(* Logix 5000 project; controller reports 1756-L63 rev 20.15; software revision 20.04; part 29 of 52 *)

        [2115].log_data[19].valid := 1, [2115].time.Year := 2023, [2115].time.Month := 1, [2115].time.Day := 17, [2115].time.Minute := 39, [2115].time.Second := 59, [2116].log_data[0].min := 1.0, [2116].log_data[0].max := 1.0, [2116].log_data[0].total := 300.0, [2116].log_data[0].time := 300.0, [2116].log_data[0].minminute := 40, [2116].log_data[0].maxminute := 40, [2116].log_data[0].valid := 1, [2116].log_data[1].valid := 1, [2116].log_data[2].valid := 1, [2116].log_data[3].valid := 1, [2116].log_data[4].valid := 1, [2116].log_data[5].valid := 1, [2116].log_data[6].valid := 1, [2116].log_data[7].valid := 1, [2116].log_data[8].valid := 1, [2116].log_data[9].valid := 1, [2116].log_data[10].valid := 1, [2116].log_data[11].valid := 1, [2116].log_data[12].valid := 1, [2116].log_data[13].valid := 1, [2116].log_data[14].valid := 1, [2116].log_data[15].valid := 1, [2116].log_data[16].valid := 1, [2116].log_data[17].valid := 1, [2116].log_data[18].valid := 1, [2116].log_data[19].valid := 1, [2116].time.Year := 2023, [2116].time.Month := 1, [2116].time.Day := 17, [2116].time.Minute := 44, [2116].time.Second := 59, [2117].log_data[0].min := 1.0, [2117].log_data[0].max := 1.0, [2117].log_data[0].total := 300.0, [2117].log_data[0].time := 300.0, [2117].log_data[0].minminute := 45, [2117].log_data[0].maxminute := 45, [2117].log_data[0].valid := 1, [2117].log_data[1].valid := 1, [2117].log_data[2].valid := 1, [2117].log_data[3].valid := 1, [2117].log_data[4].valid := 1, [2117].log_data[5].valid := 1, [2117].log_data[6].valid := 1, [2117].log_data[7].valid := 1, [2117].log_data[8].valid := 1, [2117].log_data[9].valid := 1, [2117].log_data[10].valid := 1, [2117].log_data[11].valid := 1, [2117].log_data[12].valid := 1, [2117].log_data[13].valid := 1, [2117].log_data[14].valid := 1, [2117].log_data[15].valid := 1, [2117].log_data[16].valid := 1,
        [2117].log_data[17].valid := 1, [2117].log_data[18].valid := 1, [2117].log_data[19].valid := 1, [2117].time.Year := 2023, [2117].time.Month := 1, [2117].time.Day := 17, [2117].time.Minute := 49, [2117].time.Second := 59, [2118].log_data[0].min := 1.0, [2118].log_data[0].max := 1.0, [2118].log_data[0].total := 300.0, [2118].log_data[0].time := 300.0, [2118].log_data[0].minminute := 50, [2118].log_data[0].maxminute := 50, [2118].log_data[0].valid := 1, [2118].log_data[1].valid := 1, [2118].log_data[2].valid := 1, [2118].log_data[3].valid := 1, [2118].log_data[4].valid := 1, [2118].log_data[5].valid := 1, [2118].log_data[6].valid := 1, [2118].log_data[7].valid := 1, [2118].log_data[8].valid := 1, [2118].log_data[9].valid := 1, [2118].log_data[10].valid := 1, [2118].log_data[11].valid := 1, [2118].log_data[12].valid := 1, [2118].log_data[13].valid := 1, [2118].log_data[14].valid := 1, [2118].log_data[15].valid := 1, [2118].log_data[16].valid := 1, [2118].log_data[17].valid := 1, [2118].log_data[18].valid := 1, [2118].log_data[19].valid := 1, [2118].time.Year := 2023, [2118].time.Month := 1, [2118].time.Day := 17, [2118].time.Minute := 54, [2118].time.Second := 59, [2119].log_data[0].min := 1.0, [2119].log_data[0].max := 1.0, [2119].log_data[0].total := 300.0, [2119].log_data[0].time := 300.0, [2119].log_data[0].minminute := 55, [2119].log_data[0].maxminute := 55, [2119].log_data[0].valid := 1, [2119].log_data[1].valid := 1, [2119].log_data[2].valid := 1, [2119].log_data[3].valid := 1, [2119].log_data[4].valid := 1, [2119].log_data[5].valid := 1, [2119].log_data[6].valid := 1, [2119].log_data[7].valid := 1, [2119].log_data[8].valid := 1, [2119].log_data[9].valid := 1, [2119].log_data[10].valid := 1, [2119].log_data[11].valid := 1, [2119].log_data[12].valid := 1, [2119].log_data[13].valid := 1, [2119].log_data[14].valid := 1,
        [2119].log_data[15].valid := 1, [2119].log_data[16].valid := 1, [2119].log_data[17].valid := 1, [2119].log_data[18].valid := 1, [2119].log_data[19].valid := 1, [2119].time.Year := 2023, [2119].time.Month := 1, [2119].time.Day := 17, [2119].time.Minute := 59, [2119].time.Second := 59, [2120].log_data[0].min := 1.0, [2120].log_data[0].max := 1.0, [2120].log_data[0].total := 300.0, [2120].log_data[0].time := 300.0, [2120].log_data[0].valid := 1, [2120].log_data[1].valid := 1, [2120].log_data[2].valid := 1, [2120].log_data[3].valid := 1, [2120].log_data[4].valid := 1, [2120].log_data[5].valid := 1, [2120].log_data[6].valid := 1, [2120].log_data[7].valid := 1, [2120].log_data[8].valid := 1, [2120].log_data[9].valid := 1, [2120].log_data[10].valid := 1, [2120].log_data[11].valid := 1, [2120].log_data[12].valid := 1, [2120].log_data[13].valid := 1, [2120].log_data[14].valid := 1, [2120].log_data[15].valid := 1, [2120].log_data[16].valid := 1, [2120].log_data[17].valid := 1, [2120].log_data[18].valid := 1, [2120].log_data[19].valid := 1, [2120].time.Year := 2023, [2120].time.Month := 1, [2120].time.Day := 17, [2120].time.Hour := 1, [2120].time.Minute := 4, [2120].time.Second := 59, [2121].log_data[0].min := 1.0, [2121].log_data[0].max := 1.0, [2121].log_data[0].total := 300.0, [2121].log_data[0].time := 300.0, [2121].log_data[0].minminute := 5, [2121].log_data[0].maxminute := 5, [2121].log_data[0].valid := 1, [2121].log_data[1].valid := 1, [2121].log_data[2].valid := 1, [2121].log_data[3].valid := 1, [2121].log_data[4].valid := 1, [2121].log_data[5].valid := 1, [2121].log_data[6].valid := 1, [2121].log_data[7].valid := 1, [2121].log_data[8].valid := 1, [2121].log_data[9].valid := 1, [2121].log_data[10].valid := 1, [2121].log_data[11].valid := 1, [2121].log_data[12].valid := 1, [2121].log_data[13].valid := 1,
        [2121].log_data[14].valid := 1, [2121].log_data[15].valid := 1, [2121].log_data[16].valid := 1, [2121].log_data[17].valid := 1, [2121].log_data[18].valid := 1, [2121].log_data[19].valid := 1, [2121].time.Year := 2023, [2121].time.Month := 1, [2121].time.Day := 17, [2121].time.Hour := 1, [2121].time.Minute := 9, [2121].time.Second := 59, [2122].log_data[0].min := 1.0, [2122].log_data[0].max := 1.0, [2122].log_data[0].total := 300.0, [2122].log_data[0].time := 300.0, [2122].log_data[0].minminute := 10, [2122].log_data[0].maxminute := 10, [2122].log_data[0].valid := 1, [2122].log_data[1].valid := 1, [2122].log_data[2].valid := 1, [2122].log_data[3].valid := 1, [2122].log_data[4].valid := 1, [2122].log_data[5].valid := 1, [2122].log_data[6].valid := 1, [2122].log_data[7].valid := 1, [2122].log_data[8].valid := 1, [2122].log_data[9].valid := 1, [2122].log_data[10].valid := 1, [2122].log_data[11].valid := 1, [2122].log_data[12].valid := 1, [2122].log_data[13].valid := 1, [2122].log_data[14].valid := 1, [2122].log_data[15].valid := 1, [2122].log_data[16].valid := 1, [2122].log_data[17].valid := 1, [2122].log_data[18].valid := 1, [2122].log_data[19].valid := 1, [2122].time.Year := 2023, [2122].time.Month := 1, [2122].time.Day := 17, [2122].time.Hour := 1, [2122].time.Minute := 14, [2122].time.Second := 59, [2123].log_data[0].min := 1.0, [2123].log_data[0].max := 1.0, [2123].log_data[0].total := 300.0, [2123].log_data[0].time := 300.0, [2123].log_data[0].minminute := 15, [2123].log_data[0].maxminute := 15, [2123].log_data[0].valid := 1, [2123].log_data[1].valid := 1, [2123].log_data[2].valid := 1, [2123].log_data[3].valid := 1, [2123].log_data[4].valid := 1, [2123].log_data[5].valid := 1, [2123].log_data[6].valid := 1, [2123].log_data[7].valid := 1, [2123].log_data[8].valid := 1, [2123].log_data[9].valid := 1,
        [2123].log_data[10].valid := 1, [2123].log_data[11].valid := 1, [2123].log_data[12].valid := 1, [2123].log_data[13].valid := 1, [2123].log_data[14].valid := 1, [2123].log_data[15].valid := 1, [2123].log_data[16].valid := 1, [2123].log_data[17].valid := 1, [2123].log_data[18].valid := 1, [2123].log_data[19].valid := 1, [2123].time.Year := 2023, [2123].time.Month := 1, [2123].time.Day := 17, [2123].time.Hour := 1, [2123].time.Minute := 19, [2123].time.Second := 59, [2124].log_data[0].min := 1.0, [2124].log_data[0].max := 1.0, [2124].log_data[0].total := 300.0, [2124].log_data[0].time := 300.0, [2124].log_data[0].minminute := 20, [2124].log_data[0].maxminute := 20, [2124].log_data[0].valid := 1, [2124].log_data[1].valid := 1, [2124].log_data[2].valid := 1, [2124].log_data[3].valid := 1, [2124].log_data[4].valid := 1, [2124].log_data[5].valid := 1, [2124].log_data[6].valid := 1, [2124].log_data[7].valid := 1, [2124].log_data[8].valid := 1, [2124].log_data[9].valid := 1, [2124].log_data[10].valid := 1, [2124].log_data[11].valid := 1, [2124].log_data[12].valid := 1, [2124].log_data[13].valid := 1, [2124].log_data[14].valid := 1, [2124].log_data[15].valid := 1, [2124].log_data[16].valid := 1, [2124].log_data[17].valid := 1, [2124].log_data[18].valid := 1, [2124].log_data[19].valid := 1, [2124].time.Year := 2023, [2124].time.Month := 1, [2124].time.Day := 17, [2124].time.Hour := 1, [2124].time.Minute := 24, [2124].time.Second := 59, [2125].log_data[0].min := 1.0, [2125].log_data[0].max := 1.0, [2125].log_data[0].total := 300.0, [2125].log_data[0].time := 300.0, [2125].log_data[0].minminute := 25, [2125].log_data[0].maxminute := 25, [2125].log_data[0].valid := 1, [2125].log_data[1].valid := 1, [2125].log_data[2].valid := 1, [2125].log_data[3].valid := 1, [2125].log_data[4].valid := 1, [2125].log_data[5].valid := 1,
        [2125].log_data[6].valid := 1, [2125].log_data[7].valid := 1, [2125].log_data[8].valid := 1, [2125].log_data[9].valid := 1, [2125].log_data[10].valid := 1, [2125].log_data[11].valid := 1, [2125].log_data[12].valid := 1, [2125].log_data[13].valid := 1, [2125].log_data[14].valid := 1, [2125].log_data[15].valid := 1, [2125].log_data[16].valid := 1, [2125].log_data[17].valid := 1, [2125].log_data[18].valid := 1, [2125].log_data[19].valid := 1, [2125].time.Year := 2023, [2125].time.Month := 1, [2125].time.Day := 17, [2125].time.Hour := 1, [2125].time.Minute := 29, [2125].time.Second := 59, [2126].log_data[0].min := 1.0, [2126].log_data[0].max := 1.0, [2126].log_data[0].total := 300.0, [2126].log_data[0].time := 300.0, [2126].log_data[0].minminute := 30, [2126].log_data[0].maxminute := 30, [2126].log_data[0].valid := 1, [2126].log_data[1].valid := 1, [2126].log_data[2].valid := 1, [2126].log_data[3].valid := 1, [2126].log_data[4].valid := 1, [2126].log_data[5].valid := 1, [2126].log_data[6].valid := 1, [2126].log_data[7].valid := 1, [2126].log_data[8].valid := 1, [2126].log_data[9].valid := 1, [2126].log_data[10].valid := 1, [2126].log_data[11].valid := 1, [2126].log_data[12].valid := 1, [2126].log_data[13].valid := 1, [2126].log_data[14].valid := 1, [2126].log_data[15].valid := 1, [2126].log_data[16].valid := 1, [2126].log_data[17].valid := 1, [2126].log_data[18].valid := 1, [2126].log_data[19].valid := 1, [2126].time.Year := 2023, [2126].time.Month := 1, [2126].time.Day := 17, [2126].time.Hour := 1, [2126].time.Minute := 34, [2126].time.Second := 59, [2127].log_data[0].min := 1.0, [2127].log_data[0].max := 1.0, [2127].log_data[0].total := 300.0, [2127].log_data[0].time := 300.0, [2127].log_data[0].minminute := 35, [2127].log_data[0].maxminute := 35, [2127].log_data[0].valid := 1, [2127].log_data[1].valid := 1,
        [2127].log_data[2].valid := 1, [2127].log_data[3].valid := 1, [2127].log_data[4].valid := 1, [2127].log_data[5].valid := 1, [2127].log_data[6].valid := 1, [2127].log_data[7].valid := 1, [2127].log_data[8].valid := 1, [2127].log_data[9].valid := 1, [2127].log_data[10].valid := 1, [2127].log_data[11].valid := 1, [2127].log_data[12].valid := 1, [2127].log_data[13].valid := 1, [2127].log_data[14].valid := 1, [2127].log_data[15].valid := 1, [2127].log_data[16].valid := 1, [2127].log_data[17].valid := 1, [2127].log_data[18].valid := 1, [2127].log_data[19].valid := 1, [2127].time.Year := 2023, [2127].time.Month := 1, [2127].time.Day := 17, [2127].time.Hour := 1, [2127].time.Minute := 39, [2127].time.Second := 59, [2128].log_data[0].min := 1.0, [2128].log_data[0].max := 1.0, [2128].log_data[0].total := 300.0, [2128].log_data[0].time := 300.0, [2128].log_data[0].minminute := 40, [2128].log_data[0].maxminute := 40, [2128].log_data[0].valid := 1, [2128].log_data[1].valid := 1, [2128].log_data[2].valid := 1, [2128].log_data[3].valid := 1, [2128].log_data[4].valid := 1, [2128].log_data[5].valid := 1, [2128].log_data[6].valid := 1, [2128].log_data[7].valid := 1, [2128].log_data[8].valid := 1, [2128].log_data[9].valid := 1, [2128].log_data[10].valid := 1, [2128].log_data[11].valid := 1, [2128].log_data[12].valid := 1, [2128].log_data[13].valid := 1, [2128].log_data[14].valid := 1, [2128].log_data[15].valid := 1, [2128].log_data[16].valid := 1, [2128].log_data[17].valid := 1, [2128].log_data[18].valid := 1, [2128].log_data[19].valid := 1, [2128].time.Year := 2023, [2128].time.Month := 1, [2128].time.Day := 17, [2128].time.Hour := 1, [2128].time.Minute := 44, [2128].time.Second := 59, [2129].log_data[0].min := 1.0, [2129].log_data[0].max := 1.0, [2129].log_data[0].total := 300.0, [2129].log_data[0].time := 300.0,
        [2129].log_data[0].minminute := 45, [2129].log_data[0].maxminute := 45, [2129].log_data[0].valid := 1, [2129].log_data[1].valid := 1, [2129].log_data[2].valid := 1, [2129].log_data[3].valid := 1, [2129].log_data[4].valid := 1, [2129].log_data[5].valid := 1, [2129].log_data[6].valid := 1, [2129].log_data[7].valid := 1, [2129].log_data[8].valid := 1, [2129].log_data[9].valid := 1, [2129].log_data[10].valid := 1, [2129].log_data[11].valid := 1, [2129].log_data[12].valid := 1, [2129].log_data[13].valid := 1, [2129].log_data[14].valid := 1, [2129].log_data[15].valid := 1, [2129].log_data[16].valid := 1, [2129].log_data[17].valid := 1, [2129].log_data[18].valid := 1, [2129].log_data[19].valid := 1, [2129].time.Year := 2023, [2129].time.Month := 1, [2129].time.Day := 17, [2129].time.Hour := 1, [2129].time.Minute := 49, [2129].time.Second := 59, [2130].log_data[0].min := 1.0, [2130].log_data[0].max := 1.0, [2130].log_data[0].total := 300.0, [2130].log_data[0].time := 300.0, [2130].log_data[0].minminute := 50, [2130].log_data[0].maxminute := 50, [2130].log_data[0].valid := 1, [2130].log_data[1].valid := 1, [2130].log_data[2].valid := 1, [2130].log_data[3].valid := 1, [2130].log_data[4].valid := 1, [2130].log_data[5].valid := 1, [2130].log_data[6].valid := 1, [2130].log_data[7].valid := 1, [2130].log_data[8].valid := 1, [2130].log_data[9].valid := 1, [2130].log_data[10].valid := 1, [2130].log_data[11].valid := 1, [2130].log_data[12].valid := 1, [2130].log_data[13].valid := 1, [2130].log_data[14].valid := 1, [2130].log_data[15].valid := 1, [2130].log_data[16].valid := 1, [2130].log_data[17].valid := 1, [2130].log_data[18].valid := 1, [2130].log_data[19].valid := 1, [2130].time.Year := 2023, [2130].time.Month := 1, [2130].time.Day := 17, [2130].time.Hour := 1, [2130].time.Minute := 54, [2130].time.Second := 59,
        [2131].log_data[0].min := 1.0, [2131].log_data[0].max := 1.0, [2131].log_data[0].total := 300.0, [2131].log_data[0].time := 300.0, [2131].log_data[0].minminute := 55, [2131].log_data[0].maxminute := 55, [2131].log_data[0].valid := 1, [2131].log_data[1].valid := 1, [2131].log_data[2].valid := 1, [2131].log_data[3].valid := 1, [2131].log_data[4].valid := 1, [2131].log_data[5].valid := 1, [2131].log_data[6].valid := 1, [2131].log_data[7].valid := 1, [2131].log_data[8].valid := 1, [2131].log_data[9].valid := 1, [2131].log_data[10].valid := 1, [2131].log_data[11].valid := 1, [2131].log_data[12].valid := 1, [2131].log_data[13].valid := 1, [2131].log_data[14].valid := 1, [2131].log_data[15].valid := 1, [2131].log_data[16].valid := 1, [2131].log_data[17].valid := 1, [2131].log_data[18].valid := 1, [2131].log_data[19].valid := 1, [2131].time.Year := 2023, [2131].time.Month := 1, [2131].time.Day := 17, [2131].time.Hour := 1, [2131].time.Minute := 59, [2131].time.Second := 59, [2132].log_data[0].min := 1.0, [2132].log_data[0].max := 1.0, [2132].log_data[0].total := 300.0, [2132].log_data[0].time := 300.0, [2132].log_data[0].valid := 1, [2132].log_data[1].valid := 1, [2132].log_data[2].valid := 1, [2132].log_data[3].valid := 1, [2132].log_data[4].valid := 1, [2132].log_data[5].valid := 1, [2132].log_data[6].valid := 1, [2132].log_data[7].valid := 1, [2132].log_data[8].valid := 1, [2132].log_data[9].valid := 1, [2132].log_data[10].valid := 1, [2132].log_data[11].valid := 1, [2132].log_data[12].valid := 1, [2132].log_data[13].valid := 1, [2132].log_data[14].valid := 1, [2132].log_data[15].valid := 1, [2132].log_data[16].valid := 1, [2132].log_data[17].valid := 1, [2132].log_data[18].valid := 1, [2132].log_data[19].valid := 1, [2132].time.Year := 2023, [2132].time.Month := 1, [2132].time.Day := 17, [2132].time.Hour := 2,
        [2132].time.Minute := 4, [2132].time.Second := 59, [2133].log_data[0].min := 1.0, [2133].log_data[0].max := 1.0, [2133].log_data[0].total := 300.0, [2133].log_data[0].time := 300.0, [2133].log_data[0].minminute := 5, [2133].log_data[0].maxminute := 5, [2133].log_data[0].valid := 1, [2133].log_data[1].valid := 1, [2133].log_data[2].valid := 1, [2133].log_data[3].valid := 1, [2133].log_data[4].valid := 1, [2133].log_data[5].valid := 1, [2133].log_data[6].valid := 1, [2133].log_data[7].valid := 1, [2133].log_data[8].valid := 1, [2133].log_data[9].valid := 1, [2133].log_data[10].valid := 1, [2133].log_data[11].valid := 1, [2133].log_data[12].valid := 1, [2133].log_data[13].valid := 1, [2133].log_data[14].valid := 1, [2133].log_data[15].valid := 1, [2133].log_data[16].valid := 1, [2133].log_data[17].valid := 1, [2133].log_data[18].valid := 1, [2133].log_data[19].valid := 1, [2133].time.Year := 2023, [2133].time.Month := 1, [2133].time.Day := 17, [2133].time.Hour := 2, [2133].time.Minute := 9, [2133].time.Second := 59, [2134].log_data[0].min := 1.0, [2134].log_data[0].max := 1.0, [2134].log_data[0].total := 300.0, [2134].log_data[0].time := 300.0, [2134].log_data[0].minminute := 10, [2134].log_data[0].maxminute := 10, [2134].log_data[0].valid := 1, [2134].log_data[1].valid := 1, [2134].log_data[2].valid := 1, [2134].log_data[3].valid := 1, [2134].log_data[4].valid := 1, [2134].log_data[5].valid := 1, [2134].log_data[6].valid := 1, [2134].log_data[7].valid := 1, [2134].log_data[8].valid := 1, [2134].log_data[9].valid := 1, [2134].log_data[10].valid := 1, [2134].log_data[11].valid := 1, [2134].log_data[12].valid := 1, [2134].log_data[13].valid := 1, [2134].log_data[14].valid := 1, [2134].log_data[15].valid := 1, [2134].log_data[16].valid := 1, [2134].log_data[17].valid := 1, [2134].log_data[18].valid := 1, [2134].log_data[19].valid := 1,
        [2134].time.Year := 2023, [2134].time.Month := 1, [2134].time.Day := 17, [2134].time.Hour := 2, [2134].time.Minute := 14, [2134].time.Second := 59, [2135].log_data[0].min := 1.0, [2135].log_data[0].max := 1.0, [2135].log_data[0].total := 300.0, [2135].log_data[0].time := 300.0, [2135].log_data[0].minminute := 15, [2135].log_data[0].maxminute := 15, [2135].log_data[0].valid := 1, [2135].log_data[1].valid := 1, [2135].log_data[2].valid := 1, [2135].log_data[3].valid := 1, [2135].log_data[4].valid := 1, [2135].log_data[5].valid := 1, [2135].log_data[6].valid := 1, [2135].log_data[7].valid := 1, [2135].log_data[8].valid := 1, [2135].log_data[9].valid := 1, [2135].log_data[10].valid := 1, [2135].log_data[11].valid := 1, [2135].log_data[12].valid := 1, [2135].log_data[13].valid := 1, [2135].log_data[14].valid := 1, [2135].log_data[15].valid := 1, [2135].log_data[16].valid := 1, [2135].log_data[17].valid := 1, [2135].log_data[18].valid := 1, [2135].log_data[19].valid := 1, [2135].time.Year := 2023, [2135].time.Month := 1, [2135].time.Day := 17, [2135].time.Hour := 2, [2135].time.Minute := 19, [2135].time.Second := 59, [2136].log_data[0].min := 1.0, [2136].log_data[0].max := 1.0, [2136].log_data[0].total := 300.0, [2136].log_data[0].time := 300.0, [2136].log_data[0].minminute := 20, [2136].log_data[0].maxminute := 20, [2136].log_data[0].valid := 1, [2136].log_data[1].valid := 1, [2136].log_data[2].valid := 1, [2136].log_data[3].valid := 1, [2136].log_data[4].valid := 1, [2136].log_data[5].valid := 1, [2136].log_data[6].valid := 1, [2136].log_data[7].valid := 1, [2136].log_data[8].valid := 1, [2136].log_data[9].valid := 1, [2136].log_data[10].valid := 1, [2136].log_data[11].valid := 1, [2136].log_data[12].valid := 1, [2136].log_data[13].valid := 1, [2136].log_data[14].valid := 1, [2136].log_data[15].valid := 1,
        [2136].log_data[16].valid := 1, [2136].log_data[17].valid := 1, [2136].log_data[18].valid := 1, [2136].log_data[19].valid := 1, [2136].time.Year := 2023, [2136].time.Month := 1, [2136].time.Day := 17, [2136].time.Hour := 2, [2136].time.Minute := 24, [2136].time.Second := 59, [2137].log_data[0].min := 1.0, [2137].log_data[0].max := 1.0, [2137].log_data[0].total := 300.0, [2137].log_data[0].time := 300.0, [2137].log_data[0].minminute := 25, [2137].log_data[0].maxminute := 25, [2137].log_data[0].valid := 1, [2137].log_data[1].valid := 1, [2137].log_data[2].valid := 1, [2137].log_data[3].valid := 1, [2137].log_data[4].valid := 1, [2137].log_data[5].valid := 1, [2137].log_data[6].valid := 1, [2137].log_data[7].valid := 1, [2137].log_data[8].valid := 1, [2137].log_data[9].valid := 1, [2137].log_data[10].valid := 1, [2137].log_data[11].valid := 1, [2137].log_data[12].valid := 1, [2137].log_data[13].valid := 1, [2137].log_data[14].valid := 1, [2137].log_data[15].valid := 1, [2137].log_data[16].valid := 1, [2137].log_data[17].valid := 1, [2137].log_data[18].valid := 1, [2137].log_data[19].valid := 1, [2137].time.Year := 2023, [2137].time.Month := 1, [2137].time.Day := 17, [2137].time.Hour := 2, [2137].time.Minute := 29, [2137].time.Second := 59, [2138].log_data[0].min := 1.0, [2138].log_data[0].max := 1.0, [2138].log_data[0].total := 300.0, [2138].log_data[0].time := 300.0, [2138].log_data[0].minminute := 30, [2138].log_data[0].maxminute := 30, [2138].log_data[0].valid := 1, [2138].log_data[1].valid := 1, [2138].log_data[2].valid := 1, [2138].log_data[3].valid := 1, [2138].log_data[4].valid := 1, [2138].log_data[5].valid := 1, [2138].log_data[6].valid := 1, [2138].log_data[7].valid := 1, [2138].log_data[8].valid := 1, [2138].log_data[9].valid := 1, [2138].log_data[10].valid := 1, [2138].log_data[11].valid := 1,
        [2138].log_data[12].valid := 1, [2138].log_data[13].valid := 1, [2138].log_data[14].valid := 1, [2138].log_data[15].valid := 1, [2138].log_data[16].valid := 1, [2138].log_data[17].valid := 1, [2138].log_data[18].valid := 1, [2138].log_data[19].valid := 1, [2138].time.Year := 2023, [2138].time.Month := 1, [2138].time.Day := 17, [2138].time.Hour := 2, [2138].time.Minute := 34, [2138].time.Second := 59, [2139].log_data[0].min := 1.0, [2139].log_data[0].max := 1.0, [2139].log_data[0].total := 300.0, [2139].log_data[0].time := 300.0, [2139].log_data[0].minminute := 35, [2139].log_data[0].maxminute := 35, [2139].log_data[0].valid := 1, [2139].log_data[1].valid := 1, [2139].log_data[2].valid := 1, [2139].log_data[3].valid := 1, [2139].log_data[4].valid := 1, [2139].log_data[5].valid := 1, [2139].log_data[6].valid := 1, [2139].log_data[7].valid := 1, [2139].log_data[8].valid := 1, [2139].log_data[9].valid := 1, [2139].log_data[10].valid := 1, [2139].log_data[11].valid := 1, [2139].log_data[12].valid := 1, [2139].log_data[13].valid := 1, [2139].log_data[14].valid := 1, [2139].log_data[15].valid := 1, [2139].log_data[16].valid := 1, [2139].log_data[17].valid := 1, [2139].log_data[18].valid := 1, [2139].log_data[19].valid := 1, [2139].time.Year := 2023, [2139].time.Month := 1, [2139].time.Day := 17, [2139].time.Hour := 2, [2139].time.Minute := 39, [2139].time.Second := 59, [2140].log_data[0].min := 1.0, [2140].log_data[0].max := 1.0, [2140].log_data[0].total := 300.0, [2140].log_data[0].time := 300.0, [2140].log_data[0].minminute := 40, [2140].log_data[0].maxminute := 40, [2140].log_data[0].valid := 1, [2140].log_data[1].valid := 1, [2140].log_data[2].valid := 1, [2140].log_data[3].valid := 1, [2140].log_data[4].valid := 1, [2140].log_data[5].valid := 1, [2140].log_data[6].valid := 1, [2140].log_data[7].valid := 1,
        [2140].log_data[8].valid := 1, [2140].log_data[9].valid := 1, [2140].log_data[10].valid := 1, [2140].log_data[11].valid := 1, [2140].log_data[12].valid := 1, [2140].log_data[13].valid := 1, [2140].log_data[14].valid := 1, [2140].log_data[15].valid := 1, [2140].log_data[16].valid := 1, [2140].log_data[17].valid := 1, [2140].log_data[18].valid := 1, [2140].log_data[19].valid := 1, [2140].time.Year := 2023, [2140].time.Month := 1, [2140].time.Day := 17, [2140].time.Hour := 2, [2140].time.Minute := 44, [2140].time.Second := 59, [2141].log_data[0].min := 1.0, [2141].log_data[0].max := 1.0, [2141].log_data[0].total := 300.0, [2141].log_data[0].time := 300.0, [2141].log_data[0].minminute := 45, [2141].log_data[0].maxminute := 45, [2141].log_data[0].valid := 1, [2141].log_data[1].valid := 1, [2141].log_data[2].valid := 1, [2141].log_data[3].valid := 1, [2141].log_data[4].valid := 1, [2141].log_data[5].valid := 1, [2141].log_data[6].valid := 1, [2141].log_data[7].valid := 1, [2141].log_data[8].valid := 1, [2141].log_data[9].valid := 1, [2141].log_data[10].valid := 1, [2141].log_data[11].valid := 1, [2141].log_data[12].valid := 1, [2141].log_data[13].valid := 1, [2141].log_data[14].valid := 1, [2141].log_data[15].valid := 1, [2141].log_data[16].valid := 1, [2141].log_data[17].valid := 1, [2141].log_data[18].valid := 1, [2141].log_data[19].valid := 1, [2141].time.Year := 2023, [2141].time.Month := 1, [2141].time.Day := 17, [2141].time.Hour := 2, [2141].time.Minute := 49, [2141].time.Second := 59, [2142].log_data[0].min := 1.0, [2142].log_data[0].max := 1.0, [2142].log_data[0].total := 300.0, [2142].log_data[0].time := 300.0, [2142].log_data[0].minminute := 50, [2142].log_data[0].maxminute := 50, [2142].log_data[0].valid := 1, [2142].log_data[1].valid := 1, [2142].log_data[2].valid := 1, [2142].log_data[3].valid := 1,
        [2142].log_data[4].valid := 1, [2142].log_data[5].valid := 1, [2142].log_data[6].valid := 1, [2142].log_data[7].valid := 1, [2142].log_data[8].valid := 1, [2142].log_data[9].valid := 1, [2142].log_data[10].valid := 1, [2142].log_data[11].valid := 1, [2142].log_data[12].valid := 1, [2142].log_data[13].valid := 1, [2142].log_data[14].valid := 1, [2142].log_data[15].valid := 1, [2142].log_data[16].valid := 1, [2142].log_data[17].valid := 1, [2142].log_data[18].valid := 1, [2142].log_data[19].valid := 1, [2142].time.Year := 2023, [2142].time.Month := 1, [2142].time.Day := 17, [2142].time.Hour := 2, [2142].time.Minute := 54, [2142].time.Second := 59, [2143].log_data[0].min := 1.0, [2143].log_data[0].max := 1.0, [2143].log_data[0].total := 300.0, [2143].log_data[0].time := 300.0, [2143].log_data[0].minminute := 55, [2143].log_data[0].maxminute := 55, [2143].log_data[0].valid := 1, [2143].log_data[1].valid := 1, [2143].log_data[2].valid := 1, [2143].log_data[3].valid := 1, [2143].log_data[4].valid := 1, [2143].log_data[5].valid := 1, [2143].log_data[6].valid := 1, [2143].log_data[7].valid := 1, [2143].log_data[8].valid := 1, [2143].log_data[9].valid := 1, [2143].log_data[10].valid := 1, [2143].log_data[11].valid := 1, [2143].log_data[12].valid := 1, [2143].log_data[13].valid := 1, [2143].log_data[14].valid := 1, [2143].log_data[15].valid := 1, [2143].log_data[16].valid := 1, [2143].log_data[17].valid := 1, [2143].log_data[18].valid := 1, [2143].log_data[19].valid := 1, [2143].time.Year := 2023, [2143].time.Month := 1, [2143].time.Day := 17, [2143].time.Hour := 2, [2143].time.Minute := 59, [2143].time.Second := 59, [2144].log_data[0].min := 1.0, [2144].log_data[0].max := 1.0, [2144].log_data[0].total := 300.0, [2144].log_data[0].time := 300.0, [2144].log_data[0].valid := 1, [2144].log_data[1].valid := 1,
        [2144].log_data[2].valid := 1, [2144].log_data[3].valid := 1, [2144].log_data[4].valid := 1, [2144].log_data[5].valid := 1, [2144].log_data[6].valid := 1, [2144].log_data[7].valid := 1, [2144].log_data[8].valid := 1, [2144].log_data[9].valid := 1, [2144].log_data[10].valid := 1, [2144].log_data[11].valid := 1, [2144].log_data[12].valid := 1, [2144].log_data[13].valid := 1, [2144].log_data[14].valid := 1, [2144].log_data[15].valid := 1, [2144].log_data[16].valid := 1, [2144].log_data[17].valid := 1, [2144].log_data[18].valid := 1, [2144].log_data[19].valid := 1, [2144].time.Year := 2023, [2144].time.Month := 1, [2144].time.Day := 17, [2144].time.Hour := 3, [2144].time.Minute := 4, [2144].time.Second := 59, [2145].log_data[0].min := 1.0, [2145].log_data[0].max := 1.0, [2145].log_data[0].total := 300.0, [2145].log_data[0].time := 300.0, [2145].log_data[0].minminute := 5, [2145].log_data[0].maxminute := 5, [2145].log_data[0].valid := 1, [2145].log_data[1].valid := 1, [2145].log_data[2].valid := 1, [2145].log_data[3].valid := 1, [2145].log_data[4].valid := 1, [2145].log_data[5].valid := 1, [2145].log_data[6].valid := 1, [2145].log_data[7].valid := 1, [2145].log_data[8].valid := 1, [2145].log_data[9].valid := 1, [2145].log_data[10].valid := 1, [2145].log_data[11].valid := 1, [2145].log_data[12].valid := 1, [2145].log_data[13].valid := 1, [2145].log_data[14].valid := 1, [2145].log_data[15].valid := 1, [2145].log_data[16].valid := 1, [2145].log_data[17].valid := 1, [2145].log_data[18].valid := 1, [2145].log_data[19].valid := 1, [2145].time.Year := 2023, [2145].time.Month := 1, [2145].time.Day := 17, [2145].time.Hour := 3, [2145].time.Minute := 9, [2145].time.Second := 59, [2146].log_data[0].min := 1.0, [2146].log_data[0].max := 1.0, [2146].log_data[0].total := 300.0, [2146].log_data[0].time := 300.0,
        [2146].log_data[0].minminute := 10, [2146].log_data[0].maxminute := 10, [2146].log_data[0].valid := 1, [2146].log_data[1].valid := 1, [2146].log_data[2].valid := 1, [2146].log_data[3].valid := 1, [2146].log_data[4].valid := 1, [2146].log_data[5].valid := 1, [2146].log_data[6].valid := 1, [2146].log_data[7].valid := 1, [2146].log_data[8].valid := 1, [2146].log_data[9].valid := 1, [2146].log_data[10].valid := 1, [2146].log_data[11].valid := 1, [2146].log_data[12].valid := 1, [2146].log_data[13].valid := 1, [2146].log_data[14].valid := 1, [2146].log_data[15].valid := 1, [2146].log_data[16].valid := 1, [2146].log_data[17].valid := 1, [2146].log_data[18].valid := 1, [2146].log_data[19].valid := 1, [2146].time.Year := 2023, [2146].time.Month := 1, [2146].time.Day := 17, [2146].time.Hour := 3, [2146].time.Minute := 14, [2146].time.Second := 59, [2147].log_data[0].min := 1.0, [2147].log_data[0].max := 1.0, [2147].log_data[0].total := 300.0, [2147].log_data[0].time := 300.0, [2147].log_data[0].minminute := 15, [2147].log_data[0].maxminute := 15, [2147].log_data[0].valid := 1, [2147].log_data[1].valid := 1, [2147].log_data[2].valid := 1, [2147].log_data[3].valid := 1, [2147].log_data[4].valid := 1, [2147].log_data[5].valid := 1, [2147].log_data[6].valid := 1, [2147].log_data[7].valid := 1, [2147].log_data[8].valid := 1, [2147].log_data[9].valid := 1, [2147].log_data[10].valid := 1, [2147].log_data[11].valid := 1, [2147].log_data[12].valid := 1, [2147].log_data[13].valid := 1, [2147].log_data[14].valid := 1, [2147].log_data[15].valid := 1, [2147].log_data[16].valid := 1, [2147].log_data[17].valid := 1, [2147].log_data[18].valid := 1, [2147].log_data[19].valid := 1, [2147].time.Year := 2023, [2147].time.Month := 1, [2147].time.Day := 17, [2147].time.Hour := 3, [2147].time.Minute := 19, [2147].time.Second := 59,
        [2148].log_data[0].min := 1.0, [2148].log_data[0].max := 1.0, [2148].log_data[0].total := 300.0, [2148].log_data[0].time := 300.0, [2148].log_data[0].minminute := 20, [2148].log_data[0].maxminute := 20, [2148].log_data[0].valid := 1, [2148].log_data[1].valid := 1, [2148].log_data[2].valid := 1, [2148].log_data[3].valid := 1, [2148].log_data[4].valid := 1, [2148].log_data[5].valid := 1, [2148].log_data[6].valid := 1, [2148].log_data[7].valid := 1, [2148].log_data[8].valid := 1, [2148].log_data[9].valid := 1, [2148].log_data[10].valid := 1, [2148].log_data[11].valid := 1, [2148].log_data[12].valid := 1, [2148].log_data[13].valid := 1, [2148].log_data[14].valid := 1, [2148].log_data[15].valid := 1, [2148].log_data[16].valid := 1, [2148].log_data[17].valid := 1, [2148].log_data[18].valid := 1, [2148].log_data[19].valid := 1, [2148].time.Year := 2023, [2148].time.Month := 1, [2148].time.Day := 17, [2148].time.Hour := 3, [2148].time.Minute := 24, [2148].time.Second := 59, [2149].log_data[0].min := 1.0, [2149].log_data[0].max := 1.0, [2149].log_data[0].total := 300.0, [2149].log_data[0].time := 300.0, [2149].log_data[0].minminute := 25, [2149].log_data[0].maxminute := 25, [2149].log_data[0].valid := 1, [2149].log_data[1].valid := 1, [2149].log_data[2].valid := 1, [2149].log_data[3].valid := 1, [2149].log_data[4].valid := 1, [2149].log_data[5].valid := 1, [2149].log_data[6].valid := 1, [2149].log_data[7].valid := 1, [2149].log_data[8].valid := 1, [2149].log_data[9].valid := 1, [2149].log_data[10].valid := 1, [2149].log_data[11].valid := 1, [2149].log_data[12].valid := 1, [2149].log_data[13].valid := 1, [2149].log_data[14].valid := 1, [2149].log_data[15].valid := 1, [2149].log_data[16].valid := 1, [2149].log_data[17].valid := 1, [2149].log_data[18].valid := 1, [2149].log_data[19].valid := 1, [2149].time.Year := 2023, [2149].time.Month := 1,
        [2149].time.Day := 17, [2149].time.Hour := 3, [2149].time.Minute := 29, [2149].time.Second := 59, [2150].log_data[0].min := 1.0, [2150].log_data[0].max := 1.0, [2150].log_data[0].total := 300.0, [2150].log_data[0].time := 300.0, [2150].log_data[0].minminute := 30, [2150].log_data[0].maxminute := 30, [2150].log_data[0].valid := 1, [2150].log_data[1].valid := 1, [2150].log_data[2].valid := 1, [2150].log_data[3].valid := 1, [2150].log_data[4].valid := 1, [2150].log_data[5].valid := 1, [2150].log_data[6].valid := 1, [2150].log_data[7].valid := 1, [2150].log_data[8].valid := 1, [2150].log_data[9].valid := 1, [2150].log_data[10].valid := 1, [2150].log_data[11].valid := 1, [2150].log_data[12].valid := 1, [2150].log_data[13].valid := 1, [2150].log_data[14].valid := 1, [2150].log_data[15].valid := 1, [2150].log_data[16].valid := 1, [2150].log_data[17].valid := 1, [2150].log_data[18].valid := 1, [2150].log_data[19].valid := 1, [2150].time.Year := 2023, [2150].time.Month := 1, [2150].time.Day := 17, [2150].time.Hour := 3, [2150].time.Minute := 34, [2150].time.Second := 59, [2151].log_data[0].min := 1.0, [2151].log_data[0].max := 1.0, [2151].log_data[0].total := 300.0, [2151].log_data[0].time := 300.0, [2151].log_data[0].minminute := 35, [2151].log_data[0].maxminute := 35, [2151].log_data[0].valid := 1, [2151].log_data[1].valid := 1, [2151].log_data[2].valid := 1, [2151].log_data[3].valid := 1, [2151].log_data[4].valid := 1, [2151].log_data[5].valid := 1, [2151].log_data[6].valid := 1, [2151].log_data[7].valid := 1, [2151].log_data[8].valid := 1, [2151].log_data[9].valid := 1, [2151].log_data[10].valid := 1, [2151].log_data[11].valid := 1, [2151].log_data[12].valid := 1, [2151].log_data[13].valid := 1, [2151].log_data[14].valid := 1, [2151].log_data[15].valid := 1, [2151].log_data[16].valid := 1, [2151].log_data[17].valid := 1,
        [2151].log_data[18].valid := 1, [2151].log_data[19].valid := 1, [2151].time.Year := 2023, [2151].time.Month := 1, [2151].time.Day := 17, [2151].time.Hour := 3, [2151].time.Minute := 39, [2151].time.Second := 59, [2152].log_data[0].min := 1.0, [2152].log_data[0].max := 1.0, [2152].log_data[0].total := 300.0, [2152].log_data[0].time := 300.0, [2152].log_data[0].minminute := 40, [2152].log_data[0].maxminute := 40, [2152].log_data[0].valid := 1, [2152].log_data[1].valid := 1, [2152].log_data[2].valid := 1, [2152].log_data[3].valid := 1, [2152].log_data[4].valid := 1, [2152].log_data[5].valid := 1, [2152].log_data[6].valid := 1, [2152].log_data[7].valid := 1, [2152].log_data[8].valid := 1, [2152].log_data[9].valid := 1, [2152].log_data[10].valid := 1, [2152].log_data[11].valid := 1, [2152].log_data[12].valid := 1, [2152].log_data[13].valid := 1, [2152].log_data[14].valid := 1, [2152].log_data[15].valid := 1, [2152].log_data[16].valid := 1, [2152].log_data[17].valid := 1, [2152].log_data[18].valid := 1, [2152].log_data[19].valid := 1, [2152].time.Year := 2023, [2152].time.Month := 1, [2152].time.Day := 17, [2152].time.Hour := 3, [2152].time.Minute := 44, [2152].time.Second := 59, [2153].log_data[0].min := 1.0, [2153].log_data[0].max := 1.0, [2153].log_data[0].total := 300.0, [2153].log_data[0].time := 300.0, [2153].log_data[0].minminute := 45, [2153].log_data[0].maxminute := 45, [2153].log_data[0].valid := 1, [2153].log_data[1].valid := 1, [2153].log_data[2].valid := 1, [2153].log_data[3].valid := 1, [2153].log_data[4].valid := 1, [2153].log_data[5].valid := 1, [2153].log_data[6].valid := 1, [2153].log_data[7].valid := 1, [2153].log_data[8].valid := 1, [2153].log_data[9].valid := 1, [2153].log_data[10].valid := 1, [2153].log_data[11].valid := 1, [2153].log_data[12].valid := 1, [2153].log_data[13].valid := 1,
        [2153].log_data[14].valid := 1, [2153].log_data[15].valid := 1, [2153].log_data[16].valid := 1, [2153].log_data[17].valid := 1, [2153].log_data[18].valid := 1, [2153].log_data[19].valid := 1, [2153].time.Year := 2023, [2153].time.Month := 1, [2153].time.Day := 17, [2153].time.Hour := 3, [2153].time.Minute := 49, [2153].time.Second := 59, [2154].log_data[0].min := 1.0, [2154].log_data[0].max := 1.0, [2154].log_data[0].total := 300.0, [2154].log_data[0].time := 300.0, [2154].log_data[0].minminute := 50, [2154].log_data[0].maxminute := 50, [2154].log_data[0].valid := 1, [2154].log_data[1].valid := 1, [2154].log_data[2].valid := 1, [2154].log_data[3].valid := 1, [2154].log_data[4].valid := 1, [2154].log_data[5].valid := 1, [2154].log_data[6].valid := 1, [2154].log_data[7].valid := 1, [2154].log_data[8].valid := 1, [2154].log_data[9].valid := 1, [2154].log_data[10].valid := 1, [2154].log_data[11].valid := 1, [2154].log_data[12].valid := 1, [2154].log_data[13].valid := 1, [2154].log_data[14].valid := 1, [2154].log_data[15].valid := 1, [2154].log_data[16].valid := 1, [2154].log_data[17].valid := 1, [2154].log_data[18].valid := 1, [2154].log_data[19].valid := 1, [2154].time.Year := 2023, [2154].time.Month := 1, [2154].time.Day := 17, [2154].time.Hour := 3, [2154].time.Minute := 54, [2154].time.Second := 59, [2155].log_data[0].min := 1.0, [2155].log_data[0].max := 1.0, [2155].log_data[0].total := 300.0, [2155].log_data[0].time := 300.0, [2155].log_data[0].minminute := 55, [2155].log_data[0].maxminute := 55, [2155].log_data[0].valid := 1, [2155].log_data[1].valid := 1, [2155].log_data[2].valid := 1, [2155].log_data[3].valid := 1, [2155].log_data[4].valid := 1, [2155].log_data[5].valid := 1, [2155].log_data[6].valid := 1, [2155].log_data[7].valid := 1, [2155].log_data[8].valid := 1, [2155].log_data[9].valid := 1,
        [2155].log_data[10].valid := 1, [2155].log_data[11].valid := 1, [2155].log_data[12].valid := 1, [2155].log_data[13].valid := 1, [2155].log_data[14].valid := 1, [2155].log_data[15].valid := 1, [2155].log_data[16].valid := 1, [2155].log_data[17].valid := 1, [2155].log_data[18].valid := 1, [2155].log_data[19].valid := 1, [2155].time.Year := 2023, [2155].time.Month := 1, [2155].time.Day := 17, [2155].time.Hour := 3, [2155].time.Minute := 59, [2155].time.Second := 59, [2156].log_data[0].min := 1.0, [2156].log_data[0].max := 1.0, [2156].log_data[0].total := 300.0, [2156].log_data[0].time := 300.0, [2156].log_data[0].valid := 1, [2156].log_data[1].valid := 1, [2156].log_data[2].valid := 1, [2156].log_data[3].valid := 1, [2156].log_data[4].valid := 1, [2156].log_data[5].valid := 1, [2156].log_data[6].valid := 1, [2156].log_data[7].valid := 1, [2156].log_data[8].valid := 1, [2156].log_data[9].valid := 1, [2156].log_data[10].valid := 1, [2156].log_data[11].valid := 1, [2156].log_data[12].valid := 1, [2156].log_data[13].valid := 1, [2156].log_data[14].valid := 1, [2156].log_data[15].valid := 1, [2156].log_data[16].valid := 1, [2156].log_data[17].valid := 1, [2156].log_data[18].valid := 1, [2156].log_data[19].valid := 1, [2156].time.Year := 2023, [2156].time.Month := 1, [2156].time.Day := 17, [2156].time.Hour := 4, [2156].time.Minute := 4, [2156].time.Second := 59, [2157].log_data[0].min := 1.0, [2157].log_data[0].max := 1.0, [2157].log_data[0].total := 300.0, [2157].log_data[0].time := 300.0, [2157].log_data[0].minminute := 5, [2157].log_data[0].maxminute := 5, [2157].log_data[0].valid := 1, [2157].log_data[1].valid := 1, [2157].log_data[2].valid := 1, [2157].log_data[3].valid := 1, [2157].log_data[4].valid := 1, [2157].log_data[5].valid := 1, [2157].log_data[6].valid := 1, [2157].log_data[7].valid := 1,
        [2157].log_data[8].valid := 1, [2157].log_data[9].valid := 1, [2157].log_data[10].valid := 1, [2157].log_data[11].valid := 1, [2157].log_data[12].valid := 1, [2157].log_data[13].valid := 1, [2157].log_data[14].valid := 1, [2157].log_data[15].valid := 1, [2157].log_data[16].valid := 1, [2157].log_data[17].valid := 1, [2157].log_data[18].valid := 1, [2157].log_data[19].valid := 1, [2157].time.Year := 2023, [2157].time.Month := 1, [2157].time.Day := 17, [2157].time.Hour := 4, [2157].time.Minute := 9, [2157].time.Second := 59, [2158].log_data[0].min := 1.0, [2158].log_data[0].max := 1.0, [2158].log_data[0].total := 300.0, [2158].log_data[0].time := 300.0, [2158].log_data[0].minminute := 10, [2158].log_data[0].maxminute := 10, [2158].log_data[0].valid := 1, [2158].log_data[1].valid := 1, [2158].log_data[2].valid := 1, [2158].log_data[3].valid := 1, [2158].log_data[4].valid := 1, [2158].log_data[5].valid := 1, [2158].log_data[6].valid := 1, [2158].log_data[7].valid := 1, [2158].log_data[8].valid := 1, [2158].log_data[9].valid := 1, [2158].log_data[10].valid := 1, [2158].log_data[11].valid := 1, [2158].log_data[12].valid := 1, [2158].log_data[13].valid := 1, [2158].log_data[14].valid := 1, [2158].log_data[15].valid := 1, [2158].log_data[16].valid := 1, [2158].log_data[17].valid := 1, [2158].log_data[18].valid := 1, [2158].log_data[19].valid := 1, [2158].time.Year := 2023, [2158].time.Month := 1, [2158].time.Day := 17, [2158].time.Hour := 4, [2158].time.Minute := 14, [2158].time.Second := 59, [2159].log_data[0].min := 1.0, [2159].log_data[0].max := 1.0, [2159].log_data[0].total := 300.0, [2159].log_data[0].time := 300.0, [2159].log_data[0].minminute := 15, [2159].log_data[0].maxminute := 15, [2159].log_data[0].valid := 1, [2159].log_data[1].valid := 1, [2159].log_data[2].valid := 1, [2159].log_data[3].valid := 1,
        [2159].log_data[4].valid := 1, [2159].log_data[5].valid := 1, [2159].log_data[6].valid := 1, [2159].log_data[7].valid := 1, [2159].log_data[8].valid := 1, [2159].log_data[9].valid := 1, [2159].log_data[10].valid := 1, [2159].log_data[11].valid := 1, [2159].log_data[12].valid := 1, [2159].log_data[13].valid := 1, [2159].log_data[14].valid := 1, [2159].log_data[15].valid := 1, [2159].log_data[16].valid := 1, [2159].log_data[17].valid := 1, [2159].log_data[18].valid := 1, [2159].log_data[19].valid := 1, [2159].time.Year := 2023, [2159].time.Month := 1, [2159].time.Day := 17, [2159].time.Hour := 4, [2159].time.Minute := 19, [2159].time.Second := 59, [2160].log_data[0].min := 1.0, [2160].log_data[0].max := 1.0, [2160].log_data[0].total := 300.0, [2160].log_data[0].time := 300.0, [2160].log_data[0].minminute := 20, [2160].log_data[0].maxminute := 20, [2160].log_data[0].valid := 1, [2160].log_data[1].valid := 1, [2160].log_data[2].valid := 1, [2160].log_data[3].valid := 1, [2160].log_data[4].valid := 1, [2160].log_data[5].valid := 1, [2160].log_data[6].valid := 1, [2160].log_data[7].valid := 1, [2160].log_data[8].valid := 1, [2160].log_data[9].valid := 1, [2160].log_data[10].valid := 1, [2160].log_data[11].valid := 1, [2160].log_data[12].valid := 1, [2160].log_data[13].valid := 1, [2160].log_data[14].valid := 1, [2160].log_data[15].valid := 1, [2160].log_data[16].valid := 1, [2160].log_data[17].valid := 1, [2160].log_data[18].valid := 1, [2160].log_data[19].valid := 1, [2160].time.Year := 2023, [2160].time.Month := 1, [2160].time.Day := 17, [2160].time.Hour := 4, [2160].time.Minute := 24, [2160].time.Second := 59, [2161].log_data[0].min := 1.0, [2161].log_data[0].max := 1.0, [2161].log_data[0].total := 300.0, [2161].log_data[0].time := 300.0, [2161].log_data[0].minminute := 25, [2161].log_data[0].maxminute := 25,
        [2161].log_data[0].valid := 1, [2161].log_data[1].valid := 1, [2161].log_data[2].valid := 1, [2161].log_data[3].valid := 1, [2161].log_data[4].valid := 1, [2161].log_data[5].valid := 1, [2161].log_data[6].valid := 1, [2161].log_data[7].valid := 1, [2161].log_data[8].valid := 1, [2161].log_data[9].valid := 1, [2161].log_data[10].valid := 1, [2161].log_data[11].valid := 1, [2161].log_data[12].valid := 1, [2161].log_data[13].valid := 1, [2161].log_data[14].valid := 1, [2161].log_data[15].valid := 1, [2161].log_data[16].valid := 1, [2161].log_data[17].valid := 1, [2161].log_data[18].valid := 1, [2161].log_data[19].valid := 1, [2161].time.Year := 2023, [2161].time.Month := 1, [2161].time.Day := 17, [2161].time.Hour := 4, [2161].time.Minute := 29, [2161].time.Second := 59, [2162].log_data[0].min := 1.0, [2162].log_data[0].max := 1.0, [2162].log_data[0].total := 300.0, [2162].log_data[0].time := 300.0, [2162].log_data[0].minminute := 30, [2162].log_data[0].maxminute := 30, [2162].log_data[0].valid := 1, [2162].log_data[1].valid := 1, [2162].log_data[2].valid := 1, [2162].log_data[3].valid := 1, [2162].log_data[4].valid := 1, [2162].log_data[5].valid := 1, [2162].log_data[6].valid := 1, [2162].log_data[7].valid := 1, [2162].log_data[8].valid := 1, [2162].log_data[9].valid := 1, [2162].log_data[10].valid := 1, [2162].log_data[11].valid := 1, [2162].log_data[12].valid := 1, [2162].log_data[13].valid := 1, [2162].log_data[14].valid := 1, [2162].log_data[15].valid := 1, [2162].log_data[16].valid := 1, [2162].log_data[17].valid := 1, [2162].log_data[18].valid := 1, [2162].log_data[19].valid := 1, [2162].time.Year := 2023, [2162].time.Month := 1, [2162].time.Day := 17, [2162].time.Hour := 4, [2162].time.Minute := 34, [2162].time.Second := 59, [2163].log_data[0].min := 1.0, [2163].log_data[0].max := 1.0,
        [2163].log_data[0].total := 300.0, [2163].log_data[0].time := 300.0, [2163].log_data[0].minminute := 35, [2163].log_data[0].maxminute := 35, [2163].log_data[0].valid := 1, [2163].log_data[1].valid := 1, [2163].log_data[2].valid := 1, [2163].log_data[3].valid := 1, [2163].log_data[4].valid := 1, [2163].log_data[5].valid := 1, [2163].log_data[6].valid := 1, [2163].log_data[7].valid := 1, [2163].log_data[8].valid := 1, [2163].log_data[9].valid := 1, [2163].log_data[10].valid := 1, [2163].log_data[11].valid := 1, [2163].log_data[12].valid := 1, [2163].log_data[13].valid := 1, [2163].log_data[14].valid := 1, [2163].log_data[15].valid := 1, [2163].log_data[16].valid := 1, [2163].log_data[17].valid := 1, [2163].log_data[18].valid := 1, [2163].log_data[19].valid := 1, [2163].time.Year := 2023, [2163].time.Month := 1, [2163].time.Day := 17, [2163].time.Hour := 4, [2163].time.Minute := 39, [2163].time.Second := 59, [2164].log_data[0].min := 1.0, [2164].log_data[0].max := 1.0, [2164].log_data[0].total := 300.0, [2164].log_data[0].time := 300.0, [2164].log_data[0].minminute := 40, [2164].log_data[0].maxminute := 40, [2164].log_data[0].valid := 1, [2164].log_data[1].valid := 1, [2164].log_data[2].valid := 1, [2164].log_data[3].valid := 1, [2164].log_data[4].valid := 1, [2164].log_data[5].valid := 1, [2164].log_data[6].valid := 1, [2164].log_data[7].valid := 1, [2164].log_data[8].valid := 1, [2164].log_data[9].valid := 1, [2164].log_data[10].valid := 1, [2164].log_data[11].valid := 1, [2164].log_data[12].valid := 1, [2164].log_data[13].valid := 1, [2164].log_data[14].valid := 1, [2164].log_data[15].valid := 1, [2164].log_data[16].valid := 1, [2164].log_data[17].valid := 1, [2164].log_data[18].valid := 1, [2164].log_data[19].valid := 1, [2164].time.Year := 2023, [2164].time.Month := 1, [2164].time.Day := 17, [2164].time.Hour := 4,
        [2164].time.Minute := 44, [2164].time.Second := 59, [2165].log_data[0].min := 1.0, [2165].log_data[0].max := 1.0, [2165].log_data[0].total := 300.0, [2165].log_data[0].time := 300.0, [2165].log_data[0].minminute := 45, [2165].log_data[0].maxminute := 45, [2165].log_data[0].valid := 1, [2165].log_data[1].valid := 1, [2165].log_data[2].valid := 1, [2165].log_data[3].valid := 1, [2165].log_data[4].valid := 1, [2165].log_data[5].valid := 1, [2165].log_data[6].valid := 1, [2165].log_data[7].valid := 1, [2165].log_data[8].valid := 1, [2165].log_data[9].valid := 1, [2165].log_data[10].valid := 1, [2165].log_data[11].valid := 1, [2165].log_data[12].valid := 1, [2165].log_data[13].valid := 1, [2165].log_data[14].valid := 1, [2165].log_data[15].valid := 1, [2165].log_data[16].valid := 1, [2165].log_data[17].valid := 1, [2165].log_data[18].valid := 1, [2165].log_data[19].valid := 1, [2165].time.Year := 2023, [2165].time.Month := 1, [2165].time.Day := 17, [2165].time.Hour := 4, [2165].time.Minute := 49, [2165].time.Second := 59, [2166].log_data[0].min := 1.0, [2166].log_data[0].max := 1.0, [2166].log_data[0].total := 300.0, [2166].log_data[0].time := 300.0, [2166].log_data[0].minminute := 50, [2166].log_data[0].maxminute := 50, [2166].log_data[0].valid := 1, [2166].log_data[1].valid := 1, [2166].log_data[2].valid := 1, [2166].log_data[3].valid := 1, [2166].log_data[4].valid := 1, [2166].log_data[5].valid := 1, [2166].log_data[6].valid := 1, [2166].log_data[7].valid := 1, [2166].log_data[8].valid := 1, [2166].log_data[9].valid := 1, [2166].log_data[10].valid := 1, [2166].log_data[11].valid := 1, [2166].log_data[12].valid := 1, [2166].log_data[13].valid := 1, [2166].log_data[14].valid := 1, [2166].log_data[15].valid := 1, [2166].log_data[16].valid := 1, [2166].log_data[17].valid := 1, [2166].log_data[18].valid := 1, [2166].log_data[19].valid := 1,
        [2166].time.Year := 2023, [2166].time.Month := 1, [2166].time.Day := 17, [2166].time.Hour := 4, [2166].time.Minute := 54, [2166].time.Second := 59, [2167].log_data[0].min := 1.0, [2167].log_data[0].max := 1.0, [2167].log_data[0].total := 300.0, [2167].log_data[0].time := 300.0, [2167].log_data[0].minminute := 55, [2167].log_data[0].maxminute := 55, [2167].log_data[0].valid := 1, [2167].log_data[1].valid := 1, [2167].log_data[2].valid := 1, [2167].log_data[3].valid := 1, [2167].log_data[4].valid := 1, [2167].log_data[5].valid := 1, [2167].log_data[6].valid := 1, [2167].log_data[7].valid := 1, [2167].log_data[8].valid := 1, [2167].log_data[9].valid := 1, [2167].log_data[10].valid := 1, [2167].log_data[11].valid := 1, [2167].log_data[12].valid := 1, [2167].log_data[13].valid := 1, [2167].log_data[14].valid := 1, [2167].log_data[15].valid := 1, [2167].log_data[16].valid := 1, [2167].log_data[17].valid := 1, [2167].log_data[18].valid := 1, [2167].log_data[19].valid := 1, [2167].time.Year := 2023, [2167].time.Month := 1, [2167].time.Day := 17, [2167].time.Hour := 4, [2167].time.Minute := 59, [2167].time.Second := 59, [2168].log_data[0].min := 1.0, [2168].log_data[0].max := 1.0, [2168].log_data[0].total := 300.0, [2168].log_data[0].time := 300.0, [2168].log_data[0].valid := 1, [2168].log_data[1].valid := 1, [2168].log_data[2].valid := 1, [2168].log_data[3].valid := 1, [2168].log_data[4].valid := 1, [2168].log_data[5].valid := 1, [2168].log_data[6].valid := 1, [2168].log_data[7].valid := 1, [2168].log_data[8].valid := 1, [2168].log_data[9].valid := 1, [2168].log_data[10].valid := 1, [2168].log_data[11].valid := 1, [2168].log_data[12].valid := 1, [2168].log_data[13].valid := 1, [2168].log_data[14].valid := 1, [2168].log_data[15].valid := 1, [2168].log_data[16].valid := 1, [2168].log_data[17].valid := 1,
        [2168].log_data[18].valid := 1, [2168].log_data[19].valid := 1, [2168].time.Year := 2023, [2168].time.Month := 1, [2168].time.Day := 17, [2168].time.Hour := 5, [2168].time.Minute := 4, [2168].time.Second := 59, [2169].log_data[0].min := 1.0, [2169].log_data[0].max := 1.0, [2169].log_data[0].total := 300.0, [2169].log_data[0].time := 300.0, [2169].log_data[0].minminute := 5, [2169].log_data[0].maxminute := 5, [2169].log_data[0].valid := 1, [2169].log_data[1].valid := 1, [2169].log_data[2].valid := 1, [2169].log_data[3].valid := 1, [2169].log_data[4].valid := 1, [2169].log_data[5].valid := 1, [2169].log_data[6].valid := 1, [2169].log_data[7].valid := 1, [2169].log_data[8].valid := 1, [2169].log_data[9].valid := 1, [2169].log_data[10].valid := 1, [2169].log_data[11].valid := 1, [2169].log_data[12].valid := 1, [2169].log_data[13].valid := 1, [2169].log_data[14].valid := 1, [2169].log_data[15].valid := 1, [2169].log_data[16].valid := 1, [2169].log_data[17].valid := 1, [2169].log_data[18].valid := 1, [2169].log_data[19].valid := 1, [2169].time.Year := 2023, [2169].time.Month := 1, [2169].time.Day := 17, [2169].time.Hour := 5, [2169].time.Minute := 9, [2169].time.Second := 59, [2170].log_data[0].min := 1.0, [2170].log_data[0].max := 1.0, [2170].log_data[0].total := 300.0, [2170].log_data[0].time := 300.0, [2170].log_data[0].minminute := 10, [2170].log_data[0].maxminute := 10, [2170].log_data[0].valid := 1, [2170].log_data[1].valid := 1, [2170].log_data[2].valid := 1, [2170].log_data[3].valid := 1, [2170].log_data[4].valid := 1, [2170].log_data[5].valid := 1, [2170].log_data[6].valid := 1, [2170].log_data[7].valid := 1, [2170].log_data[8].valid := 1, [2170].log_data[9].valid := 1, [2170].log_data[10].valid := 1, [2170].log_data[11].valid := 1, [2170].log_data[12].valid := 1, [2170].log_data[13].valid := 1,
        [2170].log_data[14].valid := 1, [2170].log_data[15].valid := 1, [2170].log_data[16].valid := 1, [2170].log_data[17].valid := 1, [2170].log_data[18].valid := 1, [2170].log_data[19].valid := 1, [2170].time.Year := 2023, [2170].time.Month := 1, [2170].time.Day := 17, [2170].time.Hour := 5, [2170].time.Minute := 14, [2170].time.Second := 59, [2171].log_data[0].min := 1.0, [2171].log_data[0].max := 1.0, [2171].log_data[0].total := 300.0, [2171].log_data[0].time := 300.0, [2171].log_data[0].minminute := 15, [2171].log_data[0].maxminute := 15, [2171].log_data[0].valid := 1, [2171].log_data[1].valid := 1, [2171].log_data[2].valid := 1, [2171].log_data[3].valid := 1, [2171].log_data[4].valid := 1, [2171].log_data[5].valid := 1, [2171].log_data[6].valid := 1, [2171].log_data[7].valid := 1, [2171].log_data[8].valid := 1, [2171].log_data[9].valid := 1, [2171].log_data[10].valid := 1, [2171].log_data[11].valid := 1, [2171].log_data[12].valid := 1, [2171].log_data[13].valid := 1, [2171].log_data[14].valid := 1, [2171].log_data[15].valid := 1, [2171].log_data[16].valid := 1, [2171].log_data[17].valid := 1, [2171].log_data[18].valid := 1, [2171].log_data[19].valid := 1, [2171].time.Year := 2023, [2171].time.Month := 1, [2171].time.Day := 17, [2171].time.Hour := 5, [2171].time.Minute := 19, [2171].time.Second := 59, [2172].log_data[0].min := 1.0, [2172].log_data[0].max := 1.0, [2172].log_data[0].total := 300.0, [2172].log_data[0].time := 300.0, [2172].log_data[0].minminute := 20, [2172].log_data[0].maxminute := 20, [2172].log_data[0].valid := 1, [2172].log_data[1].valid := 1, [2172].log_data[2].valid := 1, [2172].log_data[3].valid := 1, [2172].log_data[4].valid := 1, [2172].log_data[5].valid := 1, [2172].log_data[6].valid := 1, [2172].log_data[7].valid := 1, [2172].log_data[8].valid := 1, [2172].log_data[9].valid := 1,
        [2172].log_data[10].valid := 1, [2172].log_data[11].valid := 1, [2172].log_data[12].valid := 1, [2172].log_data[13].valid := 1, [2172].log_data[14].valid := 1, [2172].log_data[15].valid := 1, [2172].log_data[16].valid := 1, [2172].log_data[17].valid := 1, [2172].log_data[18].valid := 1, [2172].log_data[19].valid := 1, [2172].time.Year := 2023, [2172].time.Month := 1, [2172].time.Day := 17, [2172].time.Hour := 5, [2172].time.Minute := 24, [2172].time.Second := 59, [2173].log_data[0].min := 1.0, [2173].log_data[0].max := 1.0, [2173].log_data[0].total := 300.0, [2173].log_data[0].time := 300.0, [2173].log_data[0].minminute := 25, [2173].log_data[0].maxminute := 25, [2173].log_data[0].valid := 1, [2173].log_data[1].valid := 1, [2173].log_data[2].valid := 1, [2173].log_data[3].valid := 1, [2173].log_data[4].valid := 1, [2173].log_data[5].valid := 1, [2173].log_data[6].valid := 1, [2173].log_data[7].valid := 1, [2173].log_data[8].valid := 1, [2173].log_data[9].valid := 1, [2173].log_data[10].valid := 1, [2173].log_data[11].valid := 1, [2173].log_data[12].valid := 1, [2173].log_data[13].valid := 1, [2173].log_data[14].valid := 1, [2173].log_data[15].valid := 1, [2173].log_data[16].valid := 1, [2173].log_data[17].valid := 1, [2173].log_data[18].valid := 1, [2173].log_data[19].valid := 1, [2173].time.Year := 2023, [2173].time.Month := 1, [2173].time.Day := 17, [2173].time.Hour := 5, [2173].time.Minute := 29, [2173].time.Second := 59, [2174].log_data[0].min := 1.0, [2174].log_data[0].max := 1.0, [2174].log_data[0].total := 300.0, [2174].log_data[0].time := 300.0, [2174].log_data[0].minminute := 30, [2174].log_data[0].maxminute := 30, [2174].log_data[0].valid := 1, [2174].log_data[1].valid := 1, [2174].log_data[2].valid := 1, [2174].log_data[3].valid := 1, [2174].log_data[4].valid := 1, [2174].log_data[5].valid := 1,
        [2174].log_data[6].valid := 1, [2174].log_data[7].valid := 1, [2174].log_data[8].valid := 1, [2174].log_data[9].valid := 1, [2174].log_data[10].valid := 1, [2174].log_data[11].valid := 1, [2174].log_data[12].valid := 1, [2174].log_data[13].valid := 1, [2174].log_data[14].valid := 1, [2174].log_data[15].valid := 1, [2174].log_data[16].valid := 1, [2174].log_data[17].valid := 1, [2174].log_data[18].valid := 1, [2174].log_data[19].valid := 1, [2174].time.Year := 2023, [2174].time.Month := 1, [2174].time.Day := 17, [2174].time.Hour := 5, [2174].time.Minute := 34, [2174].time.Second := 59, [2175].log_data[0].min := 1.0, [2175].log_data[0].max := 1.0, [2175].log_data[0].total := 300.0, [2175].log_data[0].time := 300.0, [2175].log_data[0].minminute := 35, [2175].log_data[0].maxminute := 35, [2175].log_data[0].valid := 1, [2175].log_data[1].valid := 1, [2175].log_data[2].valid := 1, [2175].log_data[3].valid := 1, [2175].log_data[4].valid := 1, [2175].log_data[5].valid := 1, [2175].log_data[6].valid := 1, [2175].log_data[7].valid := 1, [2175].log_data[8].valid := 1, [2175].log_data[9].valid := 1, [2175].log_data[10].valid := 1, [2175].log_data[11].valid := 1, [2175].log_data[12].valid := 1, [2175].log_data[13].valid := 1, [2175].log_data[14].valid := 1, [2175].log_data[15].valid := 1, [2175].log_data[16].valid := 1, [2175].log_data[17].valid := 1, [2175].log_data[18].valid := 1, [2175].log_data[19].valid := 1, [2175].time.Year := 2023, [2175].time.Month := 1, [2175].time.Day := 17, [2175].time.Hour := 5, [2175].time.Minute := 39, [2175].time.Second := 59, [2176].log_data[0].min := 1.0, [2176].log_data[0].max := 1.0, [2176].log_data[0].total := 300.0, [2176].log_data[0].time := 300.0, [2176].log_data[0].minminute := 40, [2176].log_data[0].maxminute := 40, [2176].log_data[0].valid := 1, [2176].log_data[1].valid := 1,
        [2176].log_data[2].valid := 1, [2176].log_data[3].valid := 1, [2176].log_data[4].valid := 1, [2176].log_data[5].valid := 1, [2176].log_data[6].valid := 1, [2176].log_data[7].valid := 1, [2176].log_data[8].valid := 1, [2176].log_data[9].valid := 1, [2176].log_data[10].valid := 1, [2176].log_data[11].valid := 1, [2176].log_data[12].valid := 1, [2176].log_data[13].valid := 1, [2176].log_data[14].valid := 1, [2176].log_data[15].valid := 1, [2176].log_data[16].valid := 1, [2176].log_data[17].valid := 1, [2176].log_data[18].valid := 1, [2176].log_data[19].valid := 1, [2176].time.Year := 2023, [2176].time.Month := 1, [2176].time.Day := 17, [2176].time.Hour := 5, [2176].time.Minute := 44, [2176].time.Second := 59, [2177].log_data[0].min := 1.0, [2177].log_data[0].max := 1.0, [2177].log_data[0].total := 300.0, [2177].log_data[0].time := 300.0, [2177].log_data[0].minminute := 45, [2177].log_data[0].maxminute := 45, [2177].log_data[0].valid := 1, [2177].log_data[1].valid := 1, [2177].log_data[2].valid := 1, [2177].log_data[3].valid := 1, [2177].log_data[4].valid := 1, [2177].log_data[5].valid := 1, [2177].log_data[6].valid := 1, [2177].log_data[7].valid := 1, [2177].log_data[8].valid := 1, [2177].log_data[9].valid := 1, [2177].log_data[10].valid := 1, [2177].log_data[11].valid := 1, [2177].log_data[12].valid := 1, [2177].log_data[13].valid := 1, [2177].log_data[14].valid := 1, [2177].log_data[15].valid := 1, [2177].log_data[16].valid := 1, [2177].log_data[17].valid := 1, [2177].log_data[18].valid := 1, [2177].log_data[19].valid := 1, [2177].time.Year := 2023, [2177].time.Month := 1, [2177].time.Day := 17, [2177].time.Hour := 5, [2177].time.Minute := 49, [2177].time.Second := 59, [2178].log_data[0].min := 1.0, [2178].log_data[0].max := 1.0, [2178].log_data[0].total := 300.0, [2178].log_data[0].time := 300.0,
        [2178].log_data[0].minminute := 50, [2178].log_data[0].maxminute := 50, [2178].log_data[0].valid := 1, [2178].log_data[1].valid := 1, [2178].log_data[2].valid := 1, [2178].log_data[3].valid := 1, [2178].log_data[4].valid := 1, [2178].log_data[5].valid := 1, [2178].log_data[6].valid := 1, [2178].log_data[7].valid := 1, [2178].log_data[8].valid := 1, [2178].log_data[9].valid := 1, [2178].log_data[10].valid := 1, [2178].log_data[11].valid := 1, [2178].log_data[12].valid := 1, [2178].log_data[13].valid := 1, [2178].log_data[14].valid := 1, [2178].log_data[15].valid := 1, [2178].log_data[16].valid := 1, [2178].log_data[17].valid := 1, [2178].log_data[18].valid := 1, [2178].log_data[19].valid := 1, [2178].time.Year := 2023, [2178].time.Month := 1, [2178].time.Day := 17, [2178].time.Hour := 5, [2178].time.Minute := 54, [2178].time.Second := 59, [2179].log_data[0].min := 1.0, [2179].log_data[0].max := 1.0, [2179].log_data[0].total := 300.0, [2179].log_data[0].time := 300.0, [2179].log_data[0].minminute := 55, [2179].log_data[0].maxminute := 55, [2179].log_data[0].valid := 1, [2179].log_data[1].valid := 1, [2179].log_data[2].valid := 1, [2179].log_data[3].valid := 1, [2179].log_data[4].valid := 1, [2179].log_data[5].valid := 1, [2179].log_data[6].valid := 1, [2179].log_data[7].valid := 1, [2179].log_data[8].valid := 1, [2179].log_data[9].valid := 1, [2179].log_data[10].valid := 1, [2179].log_data[11].valid := 1, [2179].log_data[12].valid := 1, [2179].log_data[13].valid := 1, [2179].log_data[14].valid := 1, [2179].log_data[15].valid := 1, [2179].log_data[16].valid := 1, [2179].log_data[17].valid := 1, [2179].log_data[18].valid := 1, [2179].log_data[19].valid := 1, [2179].time.Year := 2023, [2179].time.Month := 1, [2179].time.Day := 17, [2179].time.Hour := 5, [2179].time.Minute := 59, [2179].time.Second := 59,
        [2180].log_data[0].min := 1.0, [2180].log_data[0].max := 1.0, [2180].log_data[0].total := 300.0, [2180].log_data[0].time := 300.0, [2180].log_data[0].valid := 1, [2180].log_data[1].valid := 1, [2180].log_data[2].valid := 1, [2180].log_data[3].valid := 1, [2180].log_data[4].valid := 1, [2180].log_data[5].valid := 1, [2180].log_data[6].valid := 1, [2180].log_data[7].valid := 1, [2180].log_data[8].valid := 1, [2180].log_data[9].valid := 1, [2180].log_data[10].valid := 1, [2180].log_data[11].valid := 1, [2180].log_data[12].valid := 1, [2180].log_data[13].valid := 1, [2180].log_data[14].valid := 1, [2180].log_data[15].valid := 1, [2180].log_data[16].valid := 1, [2180].log_data[17].valid := 1, [2180].log_data[18].valid := 1, [2180].log_data[19].valid := 1, [2180].time.Year := 2023, [2180].time.Month := 1, [2180].time.Day := 17, [2180].time.Hour := 6, [2180].time.Minute := 4, [2180].time.Second := 59, [2181].log_data[0].min := 1.0, [2181].log_data[0].max := 1.0, [2181].log_data[0].total := 300.0, [2181].log_data[0].time := 300.0, [2181].log_data[0].minminute := 5, [2181].log_data[0].maxminute := 5, [2181].log_data[0].valid := 1, [2181].log_data[1].valid := 1, [2181].log_data[2].valid := 1, [2181].log_data[3].valid := 1, [2181].log_data[4].valid := 1, [2181].log_data[5].valid := 1, [2181].log_data[6].valid := 1, [2181].log_data[7].valid := 1, [2181].log_data[8].valid := 1, [2181].log_data[9].valid := 1, [2181].log_data[10].valid := 1, [2181].log_data[11].valid := 1, [2181].log_data[12].valid := 1, [2181].log_data[13].valid := 1, [2181].log_data[14].valid := 1, [2181].log_data[15].valid := 1, [2181].log_data[16].valid := 1, [2181].log_data[17].valid := 1, [2181].log_data[18].valid := 1, [2181].log_data[19].valid := 1, [2181].time.Year := 2023, [2181].time.Month := 1, [2181].time.Day := 17, [2181].time.Hour := 6,
        [2181].time.Minute := 9, [2181].time.Second := 59, [2182].log_data[0].min := 1.0, [2182].log_data[0].max := 1.0, [2182].log_data[0].total := 300.0, [2182].log_data[0].time := 300.0, [2182].log_data[0].minminute := 10, [2182].log_data[0].maxminute := 10, [2182].log_data[0].valid := 1, [2182].log_data[1].valid := 1, [2182].log_data[2].valid := 1, [2182].log_data[3].valid := 1, [2182].log_data[4].valid := 1, [2182].log_data[5].valid := 1, [2182].log_data[6].valid := 1, [2182].log_data[7].valid := 1, [2182].log_data[8].valid := 1, [2182].log_data[9].valid := 1, [2182].log_data[10].valid := 1, [2182].log_data[11].valid := 1, [2182].log_data[12].valid := 1, [2182].log_data[13].valid := 1, [2182].log_data[14].valid := 1, [2182].log_data[15].valid := 1, [2182].log_data[16].valid := 1, [2182].log_data[17].valid := 1, [2182].log_data[18].valid := 1, [2182].log_data[19].valid := 1, [2182].time.Year := 2023, [2182].time.Month := 1, [2182].time.Day := 17, [2182].time.Hour := 6, [2182].time.Minute := 14, [2182].time.Second := 59, [2183].log_data[0].min := 1.0, [2183].log_data[0].max := 1.0, [2183].log_data[0].total := 300.0, [2183].log_data[0].time := 300.0, [2183].log_data[0].minminute := 15, [2183].log_data[0].maxminute := 15, [2183].log_data[0].valid := 1, [2183].log_data[1].valid := 1, [2183].log_data[2].valid := 1, [2183].log_data[3].valid := 1, [2183].log_data[4].valid := 1, [2183].log_data[5].valid := 1, [2183].log_data[6].valid := 1, [2183].log_data[7].valid := 1, [2183].log_data[8].valid := 1, [2183].log_data[9].valid := 1, [2183].log_data[10].valid := 1, [2183].log_data[11].valid := 1, [2183].log_data[12].valid := 1, [2183].log_data[13].valid := 1, [2183].log_data[14].valid := 1, [2183].log_data[15].valid := 1, [2183].log_data[16].valid := 1, [2183].log_data[17].valid := 1, [2183].log_data[18].valid := 1, [2183].log_data[19].valid := 1,
        [2183].time.Year := 2023, [2183].time.Month := 1, [2183].time.Day := 17, [2183].time.Hour := 6, [2183].time.Minute := 19, [2183].time.Second := 59, [2184].log_data[0].min := 1.0, [2184].log_data[0].max := 1.0, [2184].log_data[0].total := 300.0, [2184].log_data[0].time := 300.0, [2184].log_data[0].minminute := 20, [2184].log_data[0].maxminute := 20, [2184].log_data[0].valid := 1, [2184].log_data[1].valid := 1, [2184].log_data[2].valid := 1, [2184].log_data[3].valid := 1, [2184].log_data[4].valid := 1, [2184].log_data[5].valid := 1, [2184].log_data[6].valid := 1, [2184].log_data[7].valid := 1, [2184].log_data[8].valid := 1, [2184].log_data[9].valid := 1, [2184].log_data[10].valid := 1, [2184].log_data[11].valid := 1, [2184].log_data[12].valid := 1, [2184].log_data[13].valid := 1, [2184].log_data[14].valid := 1, [2184].log_data[15].valid := 1, [2184].log_data[16].valid := 1, [2184].log_data[17].valid := 1, [2184].log_data[18].valid := 1, [2184].log_data[19].valid := 1, [2184].time.Year := 2023, [2184].time.Month := 1, [2184].time.Day := 17, [2184].time.Hour := 6, [2184].time.Minute := 24, [2184].time.Second := 59, [2185].log_data[0].min := 1.0, [2185].log_data[0].max := 1.0, [2185].log_data[0].total := 300.0, [2185].log_data[0].time := 300.0, [2185].log_data[0].minminute := 25, [2185].log_data[0].maxminute := 25, [2185].log_data[0].valid := 1, [2185].log_data[1].valid := 1, [2185].log_data[2].valid := 1, [2185].log_data[3].valid := 1, [2185].log_data[4].valid := 1, [2185].log_data[5].valid := 1, [2185].log_data[6].valid := 1, [2185].log_data[7].valid := 1, [2185].log_data[8].valid := 1, [2185].log_data[9].valid := 1, [2185].log_data[10].valid := 1, [2185].log_data[11].valid := 1, [2185].log_data[12].valid := 1, [2185].log_data[13].valid := 1, [2185].log_data[14].valid := 1, [2185].log_data[15].valid := 1,
        [2185].log_data[16].valid := 1, [2185].log_data[17].valid := 1, [2185].log_data[18].valid := 1, [2185].log_data[19].valid := 1, [2185].time.Year := 2023, [2185].time.Month := 1, [2185].time.Day := 17, [2185].time.Hour := 6, [2185].time.Minute := 29, [2185].time.Second := 59, [2186].log_data[0].min := 1.0, [2186].log_data[0].max := 1.0, [2186].log_data[0].total := 300.0, [2186].log_data[0].time := 300.0, [2186].log_data[0].minminute := 30, [2186].log_data[0].maxminute := 30, [2186].log_data[0].valid := 1, [2186].log_data[1].valid := 1, [2186].log_data[2].valid := 1, [2186].log_data[3].valid := 1, [2186].log_data[4].valid := 1, [2186].log_data[5].valid := 1, [2186].log_data[6].valid := 1, [2186].log_data[7].valid := 1, [2186].log_data[8].valid := 1, [2186].log_data[9].valid := 1, [2186].log_data[10].valid := 1, [2186].log_data[11].valid := 1, [2186].log_data[12].valid := 1, [2186].log_data[13].valid := 1, [2186].log_data[14].valid := 1, [2186].log_data[15].valid := 1, [2186].log_data[16].valid := 1, [2186].log_data[17].valid := 1, [2186].log_data[18].valid := 1, [2186].log_data[19].valid := 1, [2186].time.Year := 2023, [2186].time.Month := 1, [2186].time.Day := 17, [2186].time.Hour := 6, [2186].time.Minute := 34, [2186].time.Second := 59, [2187].log_data[0].min := 1.0, [2187].log_data[0].max := 1.0, [2187].log_data[0].total := 300.0, [2187].log_data[0].time := 300.0, [2187].log_data[0].minminute := 35, [2187].log_data[0].maxminute := 35, [2187].log_data[0].valid := 1, [2187].log_data[1].valid := 1, [2187].log_data[2].valid := 1, [2187].log_data[3].valid := 1, [2187].log_data[4].valid := 1, [2187].log_data[5].valid := 1, [2187].log_data[6].valid := 1, [2187].log_data[7].valid := 1, [2187].log_data[8].valid := 1, [2187].log_data[9].valid := 1, [2187].log_data[10].valid := 1, [2187].log_data[11].valid := 1,
        [2187].log_data[12].valid := 1, [2187].log_data[13].valid := 1, [2187].log_data[14].valid := 1, [2187].log_data[15].valid := 1, [2187].log_data[16].valid := 1, [2187].log_data[17].valid := 1, [2187].log_data[18].valid := 1, [2187].log_data[19].valid := 1, [2187].time.Year := 2023, [2187].time.Month := 1, [2187].time.Day := 17, [2187].time.Hour := 6, [2187].time.Minute := 39, [2187].time.Second := 59, [2188].log_data[0].min := 1.0, [2188].log_data[0].max := 1.0, [2188].log_data[0].total := 300.0, [2188].log_data[0].time := 300.0, [2188].log_data[0].minminute := 40, [2188].log_data[0].maxminute := 40, [2188].log_data[0].valid := 1, [2188].log_data[1].valid := 1, [2188].log_data[2].valid := 1, [2188].log_data[3].valid := 1, [2188].log_data[4].valid := 1, [2188].log_data[5].valid := 1, [2188].log_data[6].valid := 1, [2188].log_data[7].valid := 1, [2188].log_data[8].valid := 1, [2188].log_data[9].valid := 1, [2188].log_data[10].valid := 1, [2188].log_data[11].valid := 1, [2188].log_data[12].valid := 1, [2188].log_data[13].valid := 1, [2188].log_data[14].valid := 1, [2188].log_data[15].valid := 1, [2188].log_data[16].valid := 1, [2188].log_data[17].valid := 1, [2188].log_data[18].valid := 1, [2188].log_data[19].valid := 1, [2188].time.Year := 2023, [2188].time.Month := 1, [2188].time.Day := 17, [2188].time.Hour := 6, [2188].time.Minute := 44, [2188].time.Second := 59, [2189].log_data[0].min := 1.0, [2189].log_data[0].max := 1.0, [2189].log_data[0].total := 300.0, [2189].log_data[0].time := 300.0, [2189].log_data[0].minminute := 45, [2189].log_data[0].maxminute := 45, [2189].log_data[0].valid := 1, [2189].log_data[1].valid := 1, [2189].log_data[2].valid := 1, [2189].log_data[3].valid := 1, [2189].log_data[4].valid := 1, [2189].log_data[5].valid := 1, [2189].log_data[6].valid := 1, [2189].log_data[7].valid := 1,
        [2189].log_data[8].valid := 1, [2189].log_data[9].valid := 1, [2189].log_data[10].valid := 1, [2189].log_data[11].valid := 1, [2189].log_data[12].valid := 1, [2189].log_data[13].valid := 1, [2189].log_data[14].valid := 1, [2189].log_data[15].valid := 1, [2189].log_data[16].valid := 1, [2189].log_data[17].valid := 1, [2189].log_data[18].valid := 1, [2189].log_data[19].valid := 1, [2189].time.Year := 2023, [2189].time.Month := 1, [2189].time.Day := 17, [2189].time.Hour := 6, [2189].time.Minute := 49, [2189].time.Second := 59, [2190].log_data[0].min := 1.0, [2190].log_data[0].max := 1.0, [2190].log_data[0].total := 300.0, [2190].log_data[0].time := 300.0, [2190].log_data[0].minminute := 50, [2190].log_data[0].maxminute := 50, [2190].log_data[0].valid := 1, [2190].log_data[1].valid := 1, [2190].log_data[2].valid := 1, [2190].log_data[3].valid := 1, [2190].log_data[4].valid := 1, [2190].log_data[5].valid := 1, [2190].log_data[6].valid := 1, [2190].log_data[7].valid := 1, [2190].log_data[8].valid := 1, [2190].log_data[9].valid := 1, [2190].log_data[10].valid := 1, [2190].log_data[11].valid := 1, [2190].log_data[12].valid := 1, [2190].log_data[13].valid := 1, [2190].log_data[14].valid := 1, [2190].log_data[15].valid := 1, [2190].log_data[16].valid := 1, [2190].log_data[17].valid := 1, [2190].log_data[18].valid := 1, [2190].log_data[19].valid := 1, [2190].time.Year := 2023, [2190].time.Month := 1, [2190].time.Day := 17, [2190].time.Hour := 6, [2190].time.Minute := 54, [2190].time.Second := 59, [2191].log_data[0].min := 1.0, [2191].log_data[0].max := 1.0, [2191].log_data[0].total := 300.0, [2191].log_data[0].time := 300.0, [2191].log_data[0].minminute := 55, [2191].log_data[0].maxminute := 55, [2191].log_data[0].valid := 1, [2191].log_data[1].valid := 1, [2191].log_data[2].valid := 1, [2191].log_data[3].valid := 1,
        [2191].log_data[4].valid := 1, [2191].log_data[5].valid := 1, [2191].log_data[6].valid := 1, [2191].log_data[7].valid := 1, [2191].log_data[8].valid := 1, [2191].log_data[9].valid := 1, [2191].log_data[10].valid := 1, [2191].log_data[11].valid := 1, [2191].log_data[12].valid := 1, [2191].log_data[13].valid := 1, [2191].log_data[14].valid := 1, [2191].log_data[15].valid := 1, [2191].log_data[16].valid := 1, [2191].log_data[17].valid := 1, [2191].log_data[18].valid := 1, [2191].log_data[19].valid := 1, [2191].time.Year := 2023, [2191].time.Month := 1, [2191].time.Day := 17, [2191].time.Hour := 6, [2191].time.Minute := 59, [2191].time.Second := 59, [2192].log_data[0].min := 1.0, [2192].log_data[0].max := 1.0, [2192].log_data[0].total := 300.0, [2192].log_data[0].time := 300.0, [2192].log_data[0].valid := 1, [2192].log_data[1].valid := 1, [2192].log_data[2].valid := 1, [2192].log_data[3].valid := 1, [2192].log_data[4].valid := 1, [2192].log_data[5].valid := 1, [2192].log_data[6].valid := 1, [2192].log_data[7].valid := 1, [2192].log_data[8].valid := 1, [2192].log_data[9].valid := 1, [2192].log_data[10].valid := 1, [2192].log_data[11].valid := 1, [2192].log_data[12].valid := 1, [2192].log_data[13].valid := 1, [2192].log_data[14].valid := 1, [2192].log_data[15].valid := 1, [2192].log_data[16].valid := 1, [2192].log_data[17].valid := 1, [2192].log_data[18].valid := 1, [2192].log_data[19].valid := 1, [2192].time.Year := 2023, [2192].time.Month := 1, [2192].time.Day := 17, [2192].time.Hour := 7, [2192].time.Minute := 4, [2192].time.Second := 59, [2193].log_data[0].min := 1.0, [2193].log_data[0].max := 1.0, [2193].log_data[0].total := 300.0, [2193].log_data[0].time := 300.0, [2193].log_data[0].minminute := 5, [2193].log_data[0].maxminute := 5, [2193].log_data[0].valid := 1, [2193].log_data[1].valid := 1,
        [2193].log_data[2].valid := 1, [2193].log_data[3].valid := 1, [2193].log_data[4].valid := 1, [2193].log_data[5].valid := 1, [2193].log_data[6].valid := 1, [2193].log_data[7].valid := 1, [2193].log_data[8].valid := 1, [2193].log_data[9].valid := 1, [2193].log_data[10].valid := 1, [2193].log_data[11].valid := 1, [2193].log_data[12].valid := 1, [2193].log_data[13].valid := 1, [2193].log_data[14].valid := 1, [2193].log_data[15].valid := 1, [2193].log_data[16].valid := 1, [2193].log_data[17].valid := 1, [2193].log_data[18].valid := 1, [2193].log_data[19].valid := 1, [2193].time.Year := 2023, [2193].time.Month := 1, [2193].time.Day := 17, [2193].time.Hour := 7, [2193].time.Minute := 9, [2193].time.Second := 59, [2194].log_data[0].min := 1.0, [2194].log_data[0].max := 1.0, [2194].log_data[0].total := 300.0, [2194].log_data[0].time := 300.0, [2194].log_data[0].minminute := 10, [2194].log_data[0].maxminute := 10, [2194].log_data[0].valid := 1, [2194].log_data[1].valid := 1, [2194].log_data[2].valid := 1, [2194].log_data[3].valid := 1, [2194].log_data[4].valid := 1, [2194].log_data[5].valid := 1, [2194].log_data[6].valid := 1, [2194].log_data[7].valid := 1, [2194].log_data[8].valid := 1, [2194].log_data[9].valid := 1, [2194].log_data[10].valid := 1, [2194].log_data[11].valid := 1, [2194].log_data[12].valid := 1, [2194].log_data[13].valid := 1, [2194].log_data[14].valid := 1, [2194].log_data[15].valid := 1, [2194].log_data[16].valid := 1, [2194].log_data[17].valid := 1, [2194].log_data[18].valid := 1, [2194].log_data[19].valid := 1, [2194].time.Year := 2023, [2194].time.Month := 1, [2194].time.Day := 17, [2194].time.Hour := 7, [2194].time.Minute := 14, [2194].time.Second := 59, [2195].log_data[0].min := 1.0, [2195].log_data[0].max := 1.0, [2195].log_data[0].total := 300.0, [2195].log_data[0].time := 300.0,
        [2195].log_data[0].minminute := 15, [2195].log_data[0].maxminute := 15, [2195].log_data[0].valid := 1, [2195].log_data[1].valid := 1, [2195].log_data[2].valid := 1, [2195].log_data[3].valid := 1, [2195].log_data[4].valid := 1, [2195].log_data[5].valid := 1, [2195].log_data[6].valid := 1, [2195].log_data[7].valid := 1, [2195].log_data[8].valid := 1, [2195].log_data[9].valid := 1, [2195].log_data[10].valid := 1, [2195].log_data[11].valid := 1, [2195].log_data[12].valid := 1, [2195].log_data[13].valid := 1, [2195].log_data[14].valid := 1, [2195].log_data[15].valid := 1, [2195].log_data[16].valid := 1, [2195].log_data[17].valid := 1, [2195].log_data[18].valid := 1, [2195].log_data[19].valid := 1, [2195].time.Year := 2023, [2195].time.Month := 1, [2195].time.Day := 17, [2195].time.Hour := 7, [2195].time.Minute := 19, [2195].time.Second := 59, [2196].log_data[0].min := 1.0, [2196].log_data[0].max := 1.0, [2196].log_data[0].total := 300.0, [2196].log_data[0].time := 300.0, [2196].log_data[0].minminute := 20, [2196].log_data[0].maxminute := 20, [2196].log_data[0].valid := 1, [2196].log_data[1].valid := 1, [2196].log_data[2].valid := 1, [2196].log_data[3].valid := 1, [2196].log_data[4].valid := 1, [2196].log_data[5].valid := 1, [2196].log_data[6].valid := 1, [2196].log_data[7].valid := 1, [2196].log_data[8].valid := 1, [2196].log_data[9].valid := 1, [2196].log_data[10].valid := 1, [2196].log_data[11].valid := 1, [2196].log_data[12].valid := 1, [2196].log_data[13].valid := 1, [2196].log_data[14].valid := 1, [2196].log_data[15].valid := 1, [2196].log_data[16].valid := 1, [2196].log_data[17].valid := 1, [2196].log_data[18].valid := 1, [2196].log_data[19].valid := 1, [2196].time.Year := 2023, [2196].time.Month := 1, [2196].time.Day := 17, [2196].time.Hour := 7, [2196].time.Minute := 24, [2196].time.Second := 59,
        [2197].log_data[0].min := 1.0, [2197].log_data[0].max := 1.0, [2197].log_data[0].total := 300.0, [2197].log_data[0].time := 300.0, [2197].log_data[0].minminute := 25, [2197].log_data[0].maxminute := 25, [2197].log_data[0].valid := 1, [2197].log_data[1].valid := 1, [2197].log_data[2].valid := 1, [2197].log_data[3].valid := 1, [2197].log_data[4].valid := 1, [2197].log_data[5].valid := 1, [2197].log_data[6].valid := 1, [2197].log_data[7].valid := 1, [2197].log_data[8].valid := 1, [2197].log_data[9].valid := 1, [2197].log_data[10].valid := 1, [2197].log_data[11].valid := 1, [2197].log_data[12].valid := 1, [2197].log_data[13].valid := 1, [2197].log_data[14].valid := 1, [2197].log_data[15].valid := 1, [2197].log_data[16].valid := 1, [2197].log_data[17].valid := 1, [2197].log_data[18].valid := 1, [2197].log_data[19].valid := 1, [2197].time.Year := 2023, [2197].time.Month := 1, [2197].time.Day := 17, [2197].time.Hour := 7, [2197].time.Minute := 29, [2197].time.Second := 59, [2198].log_data[0].min := 1.0, [2198].log_data[0].max := 1.0, [2198].log_data[0].total := 300.0, [2198].log_data[0].time := 300.0, [2198].log_data[0].minminute := 30, [2198].log_data[0].maxminute := 30, [2198].log_data[0].valid := 1, [2198].log_data[1].valid := 1, [2198].log_data[2].valid := 1, [2198].log_data[3].valid := 1, [2198].log_data[4].valid := 1, [2198].log_data[5].valid := 1, [2198].log_data[6].valid := 1, [2198].log_data[7].valid := 1, [2198].log_data[8].valid := 1, [2198].log_data[9].valid := 1, [2198].log_data[10].valid := 1, [2198].log_data[11].valid := 1, [2198].log_data[12].valid := 1, [2198].log_data[13].valid := 1, [2198].log_data[14].valid := 1, [2198].log_data[15].valid := 1, [2198].log_data[16].valid := 1, [2198].log_data[17].valid := 1, [2198].log_data[18].valid := 1, [2198].log_data[19].valid := 1, [2198].time.Year := 2023, [2198].time.Month := 1,
        [2198].time.Day := 17, [2198].time.Hour := 7, [2198].time.Minute := 34, [2198].time.Second := 59, [2199].log_data[0].min := 1.0, [2199].log_data[0].max := 1.0, [2199].log_data[0].total := 300.0, [2199].log_data[0].time := 300.0, [2199].log_data[0].minminute := 35, [2199].log_data[0].maxminute := 35, [2199].log_data[0].valid := 1, [2199].log_data[1].valid := 1, [2199].log_data[2].valid := 1, [2199].log_data[3].valid := 1, [2199].log_data[4].valid := 1, [2199].log_data[5].valid := 1, [2199].log_data[6].valid := 1, [2199].log_data[7].valid := 1, [2199].log_data[8].valid := 1, [2199].log_data[9].valid := 1, [2199].log_data[10].valid := 1, [2199].log_data[11].valid := 1, [2199].log_data[12].valid := 1, [2199].log_data[13].valid := 1, [2199].log_data[14].valid := 1, [2199].log_data[15].valid := 1, [2199].log_data[16].valid := 1, [2199].log_data[17].valid := 1, [2199].log_data[18].valid := 1, [2199].log_data[19].valid := 1, [2199].time.Year := 2023, [2199].time.Month := 1, [2199].time.Day := 17, [2199].time.Hour := 7, [2199].time.Minute := 39, [2199].time.Second := 59, [2200].log_data[0].min := 1.0, [2200].log_data[0].max := 1.0, [2200].log_data[0].total := 300.0, [2200].log_data[0].time := 300.0, [2200].log_data[0].minminute := 40, [2200].log_data[0].maxminute := 40, [2200].log_data[0].valid := 1, [2200].log_data[1].valid := 1, [2200].log_data[2].valid := 1, [2200].log_data[3].valid := 1, [2200].log_data[4].valid := 1, [2200].log_data[5].valid := 1, [2200].log_data[6].valid := 1, [2200].log_data[7].valid := 1, [2200].log_data[8].valid := 1, [2200].log_data[9].valid := 1, [2200].log_data[10].valid := 1, [2200].log_data[11].valid := 1, [2200].log_data[12].valid := 1, [2200].log_data[13].valid := 1, [2200].log_data[14].valid := 1, [2200].log_data[15].valid := 1, [2200].log_data[16].valid := 1, [2200].log_data[17].valid := 1,
        [2200].log_data[18].valid := 1, [2200].log_data[19].valid := 1, [2200].time.Year := 2023, [2200].time.Month := 1, [2200].time.Day := 17, [2200].time.Hour := 7, [2200].time.Minute := 44, [2200].time.Second := 59, [2201].log_data[0].min := 1.0, [2201].log_data[0].max := 1.0, [2201].log_data[0].total := 300.0, [2201].log_data[0].time := 300.0, [2201].log_data[0].minminute := 45, [2201].log_data[0].maxminute := 45, [2201].log_data[0].valid := 1, [2201].log_data[1].valid := 1, [2201].log_data[2].valid := 1, [2201].log_data[3].valid := 1, [2201].log_data[4].valid := 1, [2201].log_data[5].valid := 1, [2201].log_data[6].valid := 1, [2201].log_data[7].valid := 1, [2201].log_data[8].valid := 1, [2201].log_data[9].valid := 1, [2201].log_data[10].valid := 1, [2201].log_data[11].valid := 1, [2201].log_data[12].valid := 1, [2201].log_data[13].valid := 1, [2201].log_data[14].valid := 1, [2201].log_data[15].valid := 1, [2201].log_data[16].valid := 1, [2201].log_data[17].valid := 1, [2201].log_data[18].valid := 1, [2201].log_data[19].valid := 1, [2201].time.Year := 2023, [2201].time.Month := 1, [2201].time.Day := 17, [2201].time.Hour := 7, [2201].time.Minute := 49, [2201].time.Second := 59, [2202].log_data[0].min := 1.0, [2202].log_data[0].max := 1.0, [2202].log_data[0].total := 300.0, [2202].log_data[0].time := 300.0, [2202].log_data[0].minminute := 50, [2202].log_data[0].maxminute := 50, [2202].log_data[0].valid := 1, [2202].log_data[1].valid := 1, [2202].log_data[2].valid := 1, [2202].log_data[3].valid := 1, [2202].log_data[4].valid := 1, [2202].log_data[5].valid := 1, [2202].log_data[6].valid := 1, [2202].log_data[7].valid := 1, [2202].log_data[8].valid := 1, [2202].log_data[9].valid := 1, [2202].log_data[10].valid := 1, [2202].log_data[11].valid := 1, [2202].log_data[12].valid := 1, [2202].log_data[13].valid := 1,
        [2202].log_data[14].valid := 1, [2202].log_data[15].valid := 1, [2202].log_data[16].valid := 1, [2202].log_data[17].valid := 1, [2202].log_data[18].valid := 1, [2202].log_data[19].valid := 1, [2202].time.Year := 2023, [2202].time.Month := 1, [2202].time.Day := 17, [2202].time.Hour := 7, [2202].time.Minute := 54, [2202].time.Second := 59, [2203].log_data[0].min := 1.0, [2203].log_data[0].max := 1.0, [2203].log_data[0].total := 300.0, [2203].log_data[0].time := 300.0, [2203].log_data[0].minminute := 55, [2203].log_data[0].maxminute := 55, [2203].log_data[0].valid := 1, [2203].log_data[1].valid := 1, [2203].log_data[2].valid := 1, [2203].log_data[3].valid := 1, [2203].log_data[4].valid := 1, [2203].log_data[5].valid := 1, [2203].log_data[6].valid := 1, [2203].log_data[7].valid := 1, [2203].log_data[8].valid := 1, [2203].log_data[9].valid := 1, [2203].log_data[10].valid := 1, [2203].log_data[11].valid := 1, [2203].log_data[12].valid := 1, [2203].log_data[13].valid := 1, [2203].log_data[14].valid := 1, [2203].log_data[15].valid := 1, [2203].log_data[16].valid := 1, [2203].log_data[17].valid := 1, [2203].log_data[18].valid := 1, [2203].log_data[19].valid := 1, [2203].time.Year := 2023, [2203].time.Month := 1, [2203].time.Day := 17, [2203].time.Hour := 7, [2203].time.Minute := 59, [2203].time.Second := 59, [2204].log_data[0].min := 1.0, [2204].log_data[0].max := 1.0, [2204].log_data[0].total := 300.0, [2204].log_data[0].time := 300.0, [2204].log_data[0].valid := 1, [2204].log_data[1].valid := 1, [2204].log_data[2].valid := 1, [2204].log_data[3].valid := 1, [2204].log_data[4].valid := 1, [2204].log_data[5].valid := 1, [2204].log_data[6].valid := 1, [2204].log_data[7].valid := 1, [2204].log_data[8].valid := 1, [2204].log_data[9].valid := 1, [2204].log_data[10].valid := 1, [2204].log_data[11].valid := 1,
        [2204].log_data[12].valid := 1, [2204].log_data[13].valid := 1, [2204].log_data[14].valid := 1, [2204].log_data[15].valid := 1, [2204].log_data[16].valid := 1, [2204].log_data[17].valid := 1, [2204].log_data[18].valid := 1, [2204].log_data[19].valid := 1, [2204].time.Year := 2023, [2204].time.Month := 1, [2204].time.Day := 17, [2204].time.Hour := 8, [2204].time.Minute := 4, [2204].time.Second := 59, [2205].log_data[0].min := 1.0, [2205].log_data[0].max := 1.0, [2205].log_data[0].total := 300.0, [2205].log_data[0].time := 300.0, [2205].log_data[0].minminute := 5, [2205].log_data[0].maxminute := 5, [2205].log_data[0].valid := 1, [2205].log_data[1].valid := 1, [2205].log_data[2].valid := 1, [2205].log_data[3].valid := 1, [2205].log_data[4].valid := 1, [2205].log_data[5].valid := 1, [2205].log_data[6].valid := 1, [2205].log_data[7].valid := 1, [2205].log_data[8].valid := 1, [2205].log_data[9].valid := 1, [2205].log_data[10].valid := 1, [2205].log_data[11].valid := 1, [2205].log_data[12].valid := 1, [2205].log_data[13].valid := 1, [2205].log_data[14].valid := 1, [2205].log_data[15].valid := 1, [2205].log_data[16].valid := 1, [2205].log_data[17].valid := 1, [2205].log_data[18].valid := 1, [2205].log_data[19].valid := 1, [2205].time.Year := 2023, [2205].time.Month := 1, [2205].time.Day := 17, [2205].time.Hour := 8, [2205].time.Minute := 9, [2205].time.Second := 59, [2206].log_data[0].min := 1.0, [2206].log_data[0].max := 1.0, [2206].log_data[0].total := 300.0, [2206].log_data[0].time := 300.0, [2206].log_data[0].minminute := 10, [2206].log_data[0].maxminute := 10, [2206].log_data[0].valid := 1, [2206].log_data[1].valid := 1, [2206].log_data[2].valid := 1, [2206].log_data[3].valid := 1, [2206].log_data[4].valid := 1, [2206].log_data[5].valid := 1, [2206].log_data[6].valid := 1, [2206].log_data[7].valid := 1,
        [2206].log_data[8].valid := 1, [2206].log_data[9].valid := 1, [2206].log_data[10].valid := 1, [2206].log_data[11].valid := 1, [2206].log_data[12].valid := 1, [2206].log_data[13].valid := 1, [2206].log_data[14].valid := 1, [2206].log_data[15].valid := 1, [2206].log_data[16].valid := 1, [2206].log_data[17].valid := 1, [2206].log_data[18].valid := 1, [2206].log_data[19].valid := 1, [2206].time.Year := 2023, [2206].time.Month := 1, [2206].time.Day := 17, [2206].time.Hour := 8, [2206].time.Minute := 14, [2206].time.Second := 59, [2207].log_data[0].min := 1.0, [2207].log_data[0].max := 1.0, [2207].log_data[0].total := 300.0, [2207].log_data[0].time := 300.0, [2207].log_data[0].minminute := 15, [2207].log_data[0].maxminute := 15, [2207].log_data[0].valid := 1, [2207].log_data[1].valid := 1, [2207].log_data[2].valid := 1, [2207].log_data[3].valid := 1, [2207].log_data[4].valid := 1, [2207].log_data[5].valid := 1, [2207].log_data[6].valid := 1, [2207].log_data[7].valid := 1, [2207].log_data[8].valid := 1, [2207].log_data[9].valid := 1, [2207].log_data[10].valid := 1, [2207].log_data[11].valid := 1, [2207].log_data[12].valid := 1, [2207].log_data[13].valid := 1, [2207].log_data[14].valid := 1, [2207].log_data[15].valid := 1, [2207].log_data[16].valid := 1, [2207].log_data[17].valid := 1, [2207].log_data[18].valid := 1, [2207].log_data[19].valid := 1, [2207].time.Year := 2023, [2207].time.Month := 1, [2207].time.Day := 17, [2207].time.Hour := 8, [2207].time.Minute := 19, [2207].time.Second := 59, [2208].log_data[0].min := 1.0, [2208].log_data[0].max := 1.0, [2208].log_data[0].total := 300.0, [2208].log_data[0].time := 300.0, [2208].log_data[0].minminute := 20, [2208].log_data[0].maxminute := 20, [2208].log_data[0].valid := 1, [2208].log_data[1].valid := 1, [2208].log_data[2].valid := 1, [2208].log_data[3].valid := 1,
        [2208].log_data[4].valid := 1, [2208].log_data[5].valid := 1, [2208].log_data[6].valid := 1, [2208].log_data[7].valid := 1, [2208].log_data[8].valid := 1, [2208].log_data[9].valid := 1, [2208].log_data[10].valid := 1, [2208].log_data[11].valid := 1, [2208].log_data[12].valid := 1, [2208].log_data[13].valid := 1, [2208].log_data[14].valid := 1, [2208].log_data[15].valid := 1, [2208].log_data[16].valid := 1, [2208].log_data[17].valid := 1, [2208].log_data[18].valid := 1, [2208].log_data[19].valid := 1, [2208].time.Year := 2023, [2208].time.Month := 1, [2208].time.Day := 17, [2208].time.Hour := 8, [2208].time.Minute := 24, [2208].time.Second := 59, [2209].log_data[0].min := 1.0, [2209].log_data[0].max := 1.0, [2209].log_data[0].total := 300.0, [2209].log_data[0].time := 300.0, [2209].log_data[0].minminute := 25, [2209].log_data[0].maxminute := 25, [2209].log_data[0].valid := 1, [2209].log_data[1].valid := 1, [2209].log_data[2].valid := 1, [2209].log_data[3].valid := 1, [2209].log_data[4].valid := 1, [2209].log_data[5].valid := 1, [2209].log_data[6].valid := 1, [2209].log_data[7].valid := 1, [2209].log_data[8].valid := 1, [2209].log_data[9].valid := 1, [2209].log_data[10].valid := 1, [2209].log_data[11].valid := 1, [2209].log_data[12].valid := 1, [2209].log_data[13].valid := 1, [2209].log_data[14].valid := 1, [2209].log_data[15].valid := 1, [2209].log_data[16].valid := 1, [2209].log_data[17].valid := 1, [2209].log_data[18].valid := 1, [2209].log_data[19].valid := 1, [2209].time.Year := 2023, [2209].time.Month := 1, [2209].time.Day := 17, [2209].time.Hour := 8, [2209].time.Minute := 29, [2209].time.Second := 59, [2210].log_data[0].min := 1.0, [2210].log_data[0].max := 1.0, [2210].log_data[0].total := 300.0, [2210].log_data[0].time := 300.0, [2210].log_data[0].minminute := 30, [2210].log_data[0].maxminute := 30,
        [2210].log_data[0].valid := 1, [2210].log_data[1].valid := 1, [2210].log_data[2].valid := 1, [2210].log_data[3].valid := 1, [2210].log_data[4].valid := 1, [2210].log_data[5].valid := 1, [2210].log_data[6].valid := 1, [2210].log_data[7].valid := 1, [2210].log_data[8].valid := 1, [2210].log_data[9].valid := 1, [2210].log_data[10].valid := 1, [2210].log_data[11].valid := 1, [2210].log_data[12].valid := 1, [2210].log_data[13].valid := 1, [2210].log_data[14].valid := 1, [2210].log_data[15].valid := 1, [2210].log_data[16].valid := 1, [2210].log_data[17].valid := 1, [2210].log_data[18].valid := 1, [2210].log_data[19].valid := 1, [2210].time.Year := 2023, [2210].time.Month := 1, [2210].time.Day := 17, [2210].time.Hour := 8, [2210].time.Minute := 34, [2210].time.Second := 59, [2211].log_data[0].min := 1.0, [2211].log_data[0].max := 1.0, [2211].log_data[0].total := 300.0, [2211].log_data[0].time := 300.0, [2211].log_data[0].minminute := 35, [2211].log_data[0].maxminute := 35, [2211].log_data[0].valid := 1, [2211].log_data[1].valid := 1, [2211].log_data[2].valid := 1, [2211].log_data[3].valid := 1, [2211].log_data[4].valid := 1, [2211].log_data[5].valid := 1, [2211].log_data[6].valid := 1, [2211].log_data[7].valid := 1, [2211].log_data[8].valid := 1, [2211].log_data[9].valid := 1, [2211].log_data[10].valid := 1, [2211].log_data[11].valid := 1, [2211].log_data[12].valid := 1, [2211].log_data[13].valid := 1, [2211].log_data[14].valid := 1, [2211].log_data[15].valid := 1, [2211].log_data[16].valid := 1, [2211].log_data[17].valid := 1, [2211].log_data[18].valid := 1, [2211].log_data[19].valid := 1, [2211].time.Year := 2023, [2211].time.Month := 1, [2211].time.Day := 17, [2211].time.Hour := 8, [2211].time.Minute := 39, [2211].time.Second := 59, [2212].log_data[0].min := 1.0, [2212].log_data[0].max := 1.0,
        [2212].log_data[0].total := 300.0, [2212].log_data[0].time := 300.0, [2212].log_data[0].minminute := 40, [2212].log_data[0].maxminute := 40, [2212].log_data[0].valid := 1, [2212].log_data[1].valid := 1, [2212].log_data[2].valid := 1, [2212].log_data[3].valid := 1, [2212].log_data[4].valid := 1, [2212].log_data[5].valid := 1, [2212].log_data[6].valid := 1, [2212].log_data[7].valid := 1, [2212].log_data[8].valid := 1, [2212].log_data[9].valid := 1, [2212].log_data[10].valid := 1, [2212].log_data[11].valid := 1, [2212].log_data[12].valid := 1, [2212].log_data[13].valid := 1, [2212].log_data[14].valid := 1, [2212].log_data[15].valid := 1, [2212].log_data[16].valid := 1, [2212].log_data[17].valid := 1, [2212].log_data[18].valid := 1, [2212].log_data[19].valid := 1, [2212].time.Year := 2023, [2212].time.Month := 1, [2212].time.Day := 17, [2212].time.Hour := 8, [2212].time.Minute := 44, [2212].time.Second := 59, [2213].log_data[0].min := 1.0, [2213].log_data[0].max := 1.0, [2213].log_data[0].total := 300.0, [2213].log_data[0].time := 300.0, [2213].log_data[0].minminute := 45, [2213].log_data[0].maxminute := 45, [2213].log_data[0].valid := 1, [2213].log_data[1].valid := 1, [2213].log_data[2].valid := 1, [2213].log_data[3].valid := 1, [2213].log_data[4].valid := 1, [2213].log_data[5].valid := 1, [2213].log_data[6].valid := 1, [2213].log_data[7].valid := 1, [2213].log_data[8].valid := 1, [2213].log_data[9].valid := 1, [2213].log_data[10].valid := 1, [2213].log_data[11].valid := 1, [2213].log_data[12].valid := 1, [2213].log_data[13].valid := 1, [2213].log_data[14].valid := 1, [2213].log_data[15].valid := 1, [2213].log_data[16].valid := 1, [2213].log_data[17].valid := 1, [2213].log_data[18].valid := 1, [2213].log_data[19].valid := 1, [2213].time.Year := 2023, [2213].time.Month := 1, [2213].time.Day := 17, [2213].time.Hour := 8,
        [2213].time.Minute := 49, [2213].time.Second := 59, [2214].log_data[0].min := 1.0, [2214].log_data[0].max := 1.0, [2214].log_data[0].total := 300.0, [2214].log_data[0].time := 300.0, [2214].log_data[0].minminute := 50, [2214].log_data[0].maxminute := 50, [2214].log_data[0].valid := 1, [2214].log_data[1].valid := 1, [2214].log_data[2].valid := 1, [2214].log_data[3].valid := 1, [2214].log_data[4].valid := 1, [2214].log_data[5].valid := 1, [2214].log_data[6].valid := 1, [2214].log_data[7].valid := 1, [2214].log_data[8].valid := 1, [2214].log_data[9].valid := 1, [2214].log_data[10].valid := 1, [2214].log_data[11].valid := 1, [2214].log_data[12].valid := 1, [2214].log_data[13].valid := 1, [2214].log_data[14].valid := 1, [2214].log_data[15].valid := 1, [2214].log_data[16].valid := 1, [2214].log_data[17].valid := 1, [2214].log_data[18].valid := 1, [2214].log_data[19].valid := 1, [2214].time.Year := 2023, [2214].time.Month := 1, [2214].time.Day := 17, [2214].time.Hour := 8, [2214].time.Minute := 54, [2214].time.Second := 59, [2215].log_data[0].min := 1.0, [2215].log_data[0].max := 1.0, [2215].log_data[0].total := 300.0, [2215].log_data[0].time := 300.0, [2215].log_data[0].minminute := 55, [2215].log_data[0].maxminute := 55, [2215].log_data[0].valid := 1, [2215].log_data[1].valid := 1, [2215].log_data[2].valid := 1, [2215].log_data[3].valid := 1, [2215].log_data[4].valid := 1, [2215].log_data[5].valid := 1, [2215].log_data[6].valid := 1, [2215].log_data[7].valid := 1, [2215].log_data[8].valid := 1, [2215].log_data[9].valid := 1, [2215].log_data[10].valid := 1, [2215].log_data[11].valid := 1, [2215].log_data[12].valid := 1, [2215].log_data[13].valid := 1, [2215].log_data[14].valid := 1, [2215].log_data[15].valid := 1, [2215].log_data[16].valid := 1, [2215].log_data[17].valid := 1, [2215].log_data[18].valid := 1, [2215].log_data[19].valid := 1,
        [2215].time.Year := 2023, [2215].time.Month := 1, [2215].time.Day := 17, [2215].time.Hour := 8, [2215].time.Minute := 59, [2215].time.Second := 59, [2216].log_data[0].min := 1.0, [2216].log_data[0].max := 1.0, [2216].log_data[0].total := 299.5, [2216].log_data[0].time := 299.5, [2216].log_data[0].valid := 1, [2216].log_data[1].valid := 1, [2216].log_data[2].valid := 1, [2216].log_data[3].valid := 1, [2216].log_data[4].valid := 1, [2216].log_data[5].valid := 1, [2216].log_data[6].valid := 1, [2216].log_data[7].valid := 1, [2216].log_data[8].valid := 1, [2216].log_data[9].valid := 1, [2216].log_data[10].valid := 1, [2216].log_data[11].valid := 1, [2216].log_data[12].valid := 1, [2216].log_data[13].valid := 1, [2216].log_data[14].valid := 1, [2216].log_data[15].valid := 1, [2216].log_data[16].valid := 1, [2216].log_data[17].valid := 1, [2216].log_data[18].valid := 1, [2216].log_data[19].valid := 1, [2216].time.Year := 2023, [2216].time.Month := 1, [2216].time.Day := 17, [2216].time.Hour := 9, [2216].time.Minute := 4, [2216].time.Second := 59, [2217].log_data[0].min := 1.0, [2217].log_data[0].max := 1.0, [2217].log_data[0].total := 300.0, [2217].log_data[0].time := 300.0, [2217].log_data[0].minminute := 5, [2217].log_data[0].maxminute := 5, [2217].log_data[0].valid := 1, [2217].log_data[1].valid := 1, [2217].log_data[2].valid := 1, [2217].log_data[3].valid := 1, [2217].log_data[4].valid := 1, [2217].log_data[5].valid := 1, [2217].log_data[6].valid := 1, [2217].log_data[7].valid := 1, [2217].log_data[8].valid := 1, [2217].log_data[9].valid := 1, [2217].log_data[10].valid := 1, [2217].log_data[11].valid := 1, [2217].log_data[12].valid := 1, [2217].log_data[13].valid := 1, [2217].log_data[14].valid := 1, [2217].log_data[15].valid := 1, [2217].log_data[16].valid := 1, [2217].log_data[17].valid := 1,
